													CoorFinaleLado_Pri0_Des180[NuPieza_B].LadoB.CoordenadaFinale_X := Supporto.XDim/2 + Supporto.OFSDE_X180;;
													CoorFinaleLado_Pri0_Des180[NuPieza_B].LadoB.CoordenadaFinale_Y := YEsternoLastra_A_B[NuPieza_B].Lado_B_180Grados + Supporto.OFSDE_Y0;
													CoorFinaleLado_Pri0_Des180[NuPieza_B].LadoB.CoordenadaFinale_Z := ZEsternoLastra_A_B[NuPieza_B].Lado_B_180Grados + Supporto.OFSDE_Z0;
													CoorFinaleLado_Pri0_Des180[NuPieza_B].LadoB.CoordenadaFinale_J := AlgoloAlfa_gradi + Supporto.OFSDE_J0 ;
											END_CASE
										4:	
											CASE LadoRegistarFor OF
												0: 
													CoorFinaleLado_Pri0_Des180[NuPieza_A].LadoA.CoordenadaFinale_X := Supporto.XDim/2 + Supporto.OFSDE_X0;;
													CoorFinaleLado_Pri0_Des180[NuPieza_A].LadoA.CoordenadaFinale_Y := YCoordinataAppoggioLastra_A_B[NuPieza_A].Lado_A_0Grados + Supporto.OFSDE_Y0;
													CoorFinaleLado_Pri0_Des180[NuPieza_A].LadoA.CoordenadaFinale_Z := ZCoordinataAppoggioLastra_A_B[NuPieza_A].Lado_A_0Grados + Supporto.OFSDE_Z0;
													CoorFinaleLado_Pri0_Des180[NuPieza_A].LadoA.CoordenadaFinale_J := AlgoloAlfa_gradi + Supporto.OFSDE_J0 ;
												180 :
													 
													CoorFinaleLado_Pri0_Des180[NuPieza_B].LadoB.CoordenadaFinale_X := Supporto.XDim/2 + Supporto.OFSDE_X180;;
													CoorFinaleLado_Pri0_Des180[NuPieza_B].LadoB.CoordenadaFinale_Y := YCoordinataAppoggioLastra_A_B[NuPieza_B].Lado_B_180Grados + Supporto.OFSDE_Y0;
													CoorFinaleLado_Pri0_Des180[NuPieza_B].LadoB.CoordenadaFinale_Z := ZCoordinataAppoggioLastra_A_B[NuPieza_B].Lado_B_180Grados + Supporto.OFSDE_Z0;
													CoorFinaleLado_Pri0_Des180[NuPieza_B].LadoB.CoordenadaFinale_J := AlgoloAlfa_gradi + Supporto.OFSDE_J0 ;
											END_CASE
																					
								END_CASE
										
						END_IF
					END_FOR
					
{endregion}

{Region "Ordinamento consecutivo prima un lato poi l'altro"}


		(* Ordinamento consecutivo prima un lato poi l'altro *)
		2:
			FOR Contador :=1 TO numeroLastre_int BY 1 DO
				Fun_PiezaLadoCaballete(Nu_PiezaGlobal:= Contador , Grados:= ADR(LadoRegistarFor)  ,
										 Nu_pieza_LadoA=>NuPieza_A , Nu_pieza_LadoB=> NuPieza_B  );
				IF NOT CalculoEstacionPickinPiezasDiferentes THEN 
					CASE TipoRisultato OF 
							1:	
								
								CoorFinaleLado_Pri0_Des180[Contador].LadoA.CoordenadaFinale_Y := YInternoLastra[Contador] + Supporto.OFSDE_Y0;
								CoorFinaleLado_Pri0_Des180[Contador].LadoA.CoordenadaFinale_Z := ZInternoLastra[Contador] + Supporto.OFSDE_Z0;
								
								CoorFinaleLado_Pri0_Des180[Contador].LadoB.CoordenadaFinale_Y := -YInternoLastra[Contador] + Supporto.OFSDE_Y180;
								CoorFinaleLado_Pri0_Des180[Contador].LadoB.CoordenadaFinale_Z := ZInternoLastra[Contador] + Supporto.OFSDE_Z180;
								
									
	
							2:
								CoorFinaleLado_Pri0_Des180[Contador].LadoA.CoordenadaFinale_Y := YCentroLastra[Contador] + Supporto.OFSDE_Y0;
								CoorFinaleLado_Pri0_Des180[Contador].LadoA.CoordenadaFinale_Z := ZCentroLastra[Contador] + Supporto.OFSDE_Z0;
								
								CoorFinaleLado_Pri0_Des180[Contador].LadoB.CoordenadaFinale_Y := -YCentroLastra[Contador] + Supporto.OFSDE_Y180;
								CoorFinaleLado_Pri0_Des180[Contador].LadoB.CoordenadaFinale_Z := ZCentroLastra[Contador] + Supporto.OFSDE_Z180;
							
							3:
								CoorFinaleLado_Pri0_Des180[Contador].LadoA.CoordenadaFinale_Y := YEsternoLastra[Contador] + Supporto.OFSDE_Y0;
								CoorFinaleLado_Pri0_Des180[Contador].LadoA.CoordenadaFinale_Z := ZEsternoLastra[Contador] + Supporto.OFSDE_Z0;
								
								CoorFinaleLado_Pri0_Des180[Contador].LadoB.CoordenadaFinale_Y := -YEsternoLastra[Contador] + Supporto.OFSDE_Y180;
								CoorFinaleLado_Pri0_Des180[Contador].LadoB.CoordenadaFinale_Z := ZEsternoLastra[Contador] + Supporto.OFSDE_Z180;
							
							4:
								CoorFinaleLado_Pri0_Des180[Contador].LadoA.CoordenadaFinale_Y := YCoordinataAppoggioLastra[Contador] + Supporto.OFSDE_Y0;
								CoorFinaleLado_Pri0_Des180[Contador].LadoA.CoordenadaFinale_Z := ZEsternoLastra[Contador] + Supporto.OFSDE_Z0;
								
								CoorFinaleLado_Pri0_Des180[Contador].LadoB.CoordenadaFinale_Y := -YCoordinataAppoggioLastra[Contador] + Supporto.OFSDE_Y180;
								CoorFinaleLado_Pri0_Des180[Contador].LadoB.CoordenadaFinale_Z := ZEsternoLastra[Contador] + Supporto.OFSDE_Z180;
	
					END_CASE
					CoorFinaleLado_Pri0_Des180[Contador].LadoA.CoordenadaFinale_X := Supporto.XDim/2 + Supporto.OFSDE_X180;
					CoorFinaleLado_Pri0_Des180[Contador].LadoA.CoordenadaFinale_J :=  AlgoloAlfa_gradi + Supporto.OFSDE_J0;
					CoorFinaleLado_Pri0_Des180[Contador].LadoB.CoordenadaFinale_J := 180 - AlgoloAlfa_gradi + Supporto.OFSDE_J180;
				ELSIF  CalculoEstacionPickinPiezasDiferentes AND Supporto.Tipologia = CAVALLETTO  THEN 	
					
					CASE TipoRisultato OF
						1:
							CASE LadoRegistarFor OF
								0:
									CoorFinaleLado_Pri0_Des180[NuPieza_A].LadoA.CoordenadaFinale_X := Supporto.XDim/2 + Supporto.OFSDE_X180;
									CoorFinaleLado_Pri0_Des180[NuPieza_A].LadoA.CoordenadaFinale_Y := YInternoLastra_A_B[NuPieza_A].Lado_A_0Grados + Supporto.OFSDE_Y0;
									CoorFinaleLado_Pri0_Des180[NuPieza_A].LadoA.CoordenadaFinale_Z := ZInternoLastra_A_B[NuPieza_A].Lado_A_0Grados + Supporto.OFSDE_Z0;
									CoorFinaleLado_Pri0_Des180[NuPieza_A].LadoA.CoordenadaFinale_J := AlgoloAlfa_gradi + Supporto.OFSDE_J0;
									
								180:
									CoorFinaleLado_Pri0_Des180[NuPieza_B].LadoA.CoordenadaFinale_X := Supporto.XDim/2 + Supporto.OFSDE_X180;
									CoorFinaleLado_Pri0_Des180[NuPieza_B].LadoB.CoordenadaFinale_Y := -YInternoLastra_A_B[NuPieza_B].Lado_B_180Grados + Supporto.OFSDE_Y180;
									CoorFinaleLado_Pri0_Des180[NuPieza_B].LadoB.CoordenadaFinale_Z := ZInternoLastra_A_B[NuPieza_B].Lado_B_180Grados + Supporto.OFSDE_Z180;
									CoorFinaleLado_Pri0_Des180[NuPieza_B].LadoB.CoordenadaFinale_J := 180 - AlgoloAlfa_gradi + Supporto.OFSDE_J180;
							END_CASE
						
						
						2:
							CASE LadoRegistarFor OF
								0:
									CoorFinaleLado_Pri0_Des180[NuPieza_A].LadoA.CoordenadaFinale_X := Supporto.XDim/2 + Supporto.OFSDE_X180;
									CoorFinaleLado_Pri0_Des180[NuPieza_A].LadoA.CoordenadaFinale_Y := YCentroLastra_A_B[NuPieza_A].Lado_A_0Grados + Supporto.OFSDE_Y0;
									CoorFinaleLado_Pri0_Des180[NuPieza_A].LadoA.CoordenadaFinale_Z := ZCentroLastra_A_B[NuPieza_A].Lado_A_0Grados + Supporto.OFSDE_Z0;
									CoorFinaleLado_Pri0_Des180[NuPieza_A].LadoA.CoordenadaFinale_J := AlgoloAlfa_gradi + Supporto.OFSDE_J0;
								180:
									CoorFinaleLado_Pri0_Des180[NuPieza_B].LadoA.CoordenadaFinale_X := Supporto.XDim/2 + Supporto.OFSDE_X180;
									CoorFinaleLado_Pri0_Des180[NuPieza_B].LadoB.CoordenadaFinale_Y := -YCentroLastra_A_B[NuPieza_B].Lado_B_180Grados + Supporto.OFSDE_Y180;
									CoorFinaleLado_Pri0_Des180[NuPieza_B].LadoB.CoordenadaFinale_Z := ZCentroLastra_A_B[NuPieza_B].Lado_B_180Grados + Supporto.OFSDE_Z180;
									CoorFinaleLado_Pri0_Des180[NuPieza_B].LadoB.CoordenadaFinale_J := 180 - AlgoloAlfa_gradi + Supporto.OFSDE_J180;
							END_CASE
						3:
							CASE LadoRegistarFor OF
								0:
									CoorFinaleLado_Pri0_Des180[NuPieza_A].LadoA.CoordenadaFinale_X := Supporto.XDim/2 + Supporto.OFSDE_X180;
									CoorFinaleLado_Pri0_Des180[NuPieza_A].LadoA.CoordenadaFinale_Y := YEsternoLastra_A_B[NuPieza_A].Lado_A_0Grados + Supporto.OFSDE_Y0;
									CoorFinaleLado_Pri0_Des180[NuPieza_A].LadoA.CoordenadaFinale_Z := ZEsternoLastra_A_B[NuPieza_A].Lado_A_0Grados + Supporto.OFSDE_Z0;
									CoorFinaleLado_Pri0_Des180[NuPieza_A].LadoA.CoordenadaFinale_J := AlgoloAlfa_gradi + Supporto.OFSDE_J0;
								180:
									CoorFinaleLado_Pri0_Des180[NuPieza_B].LadoA.CoordenadaFinale_X := Supporto.XDim/2 + Supporto.OFSDE_X180;
									CoorFinaleLado_Pri0_Des180[NuPieza_B].LadoB.CoordenadaFinale_Y := -YEsternoLastra_A_B[NuPieza_B].Lado_B_180Grados + Supporto.OFSDE_Y180;
									CoorFinaleLado_Pri0_Des180[NuPieza_B].LadoB.CoordenadaFinale_Z := ZEsternoLastra_A_B[NuPieza_B].Lado_B_180Grados + Supporto.OFSDE_Z180;
									CoorFinaleLado_Pri0_Des180[NuPieza_B].LadoB.CoordenadaFinale_J := 180 - AlgoloAlfa_gradi + Supporto.OFSDE_J180;
							END_CASE
						4:
							CASE LadoRegistarFor OF
								0:
									CoorFinaleLado_Pri0_Des180[NuPieza_A].LadoA.CoordenadaFinale_X := Supporto.XDim/2 + Supporto.OFSDE_X180;
									CoorFinaleLado_Pri0_Des180[NuPieza_A].LadoA.CoordenadaFinale_Y := YCoordinataAppoggioLastra_A_B[NuPieza_A].Lado_A_0Grados + Supporto.OFSDE_Y0;
									CoorFinaleLado_Pri0_Des180[NuPieza_A].LadoA.CoordenadaFinale_Z := ZEsternoLastra_A_B[NuPieza_A].Lado_A_0Grados + Supporto.OFSDE_Z0;
									CoorFinaleLado_Pri0_Des180[NuPieza_A].LadoA.CoordenadaFinale_J := AlgoloAlfa_gradi + Supporto.OFSDE_J0;
								180:
									CoorFinaleLado_Pri0_Des180[NuPieza_B].LadoA.CoordenadaFinale_X := Supporto.XDim/2 + Supporto.OFSDE_X180;
									CoorFinaleLado_Pri0_Des180[NuPieza_B].LadoB.CoordenadaFinale_Y := -YCoordinataAppoggioLastra_A_B[NuPieza_B].Lado_B_180Grados + Supporto.OFSDE_Y180;
									CoorFinaleLado_Pri0_Des180[NuPieza_B].LadoB.CoordenadaFinale_Z := ZEsternoLastra_A_B[NuPieza_B].Lado_B_180Grados + Supporto.OFSDE_Z180;
									CoorFinaleLado_Pri0_Des180[NuPieza_B].LadoB.CoordenadaFinale_J := 180 - AlgoloAlfa_gradi + Supporto.OFSDE_J180;
							END_CASE
						
						
						
						
						
					END_CASE
				
				END_IF
				END_FOR
		3:
			FOR Contador:=1 TO numeroLastre_int BY 1 DO
				XFinaleLado_0Grados[Contador] := Supporto.XDim/2 + Supporto.OFSDE_X0;
				CoorFinaleLado_Pri0_Des180[Contador].LadoA.CoordenadaFinale_X := XFinaleLado_0Grados[Contador];
					IF  NOT CalculoEstacionPickinPiezasDiferentes	THEN	
						CASE TipoRisultato OF
							1:	
								YFinaleLado_0Grados[Contador] := YInternoLastra[Contador] + Supporto.OFSDE_Y0;
								ZFinaleLado_0Grados[Contador] := ZInternoLastra[Contador] + Supporto.OFSDE_Z0;
								
							2:	
								YFinaleLado_0Grados[Contador] := YCentroLastra[Contador] + Supporto.OFSDE_Y0;
								ZFinaleLado_0Grados[Contador] := ZCentroLastra[Contador] + Supporto.OFSDE_Z0;
							3:	
								YFinaleLado_0Grados[Contador] := YEsternoLastra[Contador] + Supporto.OFSDE_Y0;
								ZFinaleLado_0Grados[Contador] := ZEsternoLastra[Contador] + Supporto.OFSDE_Z0;
							4:	
								YFinaleLado_0Grados[Contador] := YCoordinataAppoggioLastra[Contador] + Supporto.OFSDE_Y0;
								ZFinaleLado_0Grados[Contador] := ZEsternoLastra[Contador] + Supporto.OFSDE_Z0;
						END_CASE
					ELSIF CalculoEstacionPickinPiezasDiferentes	THEN
						CASE TipoRisultato OF
							1:	
								YFinaleLado_0Grados[Contador] := YInternoLastra_A_B[Contador].Lado_A_0Grados + Supporto.OFSDE_Y0;
								ZFinaleLado_0Grados[Contador] := ZInternoLastra_A_B[Contador].Lado_A_0Grados + Supporto.OFSDE_Z0;	
								
							2:	
								
								YFinaleLado_0Grados[Contador] := YCentroLastra_A_B[Contador].Lado_A_0Grados + Supporto.OFSDE_Y0;
								ZFinaleLado_0Grados[Contador] := ZCentroLastra_A_B[Contador].Lado_A_0Grados + Supporto.OFSDE_Z0;
							3:	
								YFinaleLado_0Grados[Contador] := YEsternoLastra_A_B[Contador].Lado_A_0Grados + Supporto.OFSDE_Y0;
								ZFinaleLado_0Grados[Contador] := ZEsternoLastra_A_B[Contador].Lado_A_0Grados + Supporto.OFSDE_Z0;
							4:	
								YFinaleLado_0Grados[Contador] := YCoordinataAppoggioLastra_A_B[Contador].Lado_A_0Grados + Supporto.OFSDE_Y0;
								ZFinaleLado_0Grados[Contador] := ZEsternoLastra_A_B[Contador].Lado_A_0Grados + Supporto.OFSDE_Z0;
						END_CASE
						CoorFinaleLado_Pri0_Des180[Contador].LadoA.CoordenadaFinale_Y := YFinaleLado_0Grados[Contador];	
						CoorFinaleLado_Pri0_Des180[Contador].LadoA.CoordenadaFinale_Z := ZFinaleLado_0Grados[Contador] ;
					END_IF
				
				JFinaleLado_0Grados[Contador] := AlgoloAlfa_gradi + Supporto.OFSDE_J0;
				CoorFinaleLado_Pri0_Des180[Contador].LadoA.CoordenadaFinale_J := JFinaleLado_0Grados[Contador] ;
			END_FOR	
		IF  CalculoEstacionPickinPiezasDiferentes OR NOT  HabiCalTodasCordenadas  THEN
				XFinale := 	XFinaleLado_0Grados ;	
				YFinale := 	YFinaleLado_0Grados ;
				ZFinale := 	ZFinaleLado_0Grados ;
				JFinale := 	JFinaleLado_0Grados ;	
		END_IF		
				
	4:
		FOR Contador:=1 TO numeroLastre_int BY 1 DO
						
			XFinaleLado_180Grados[Contador] := Supporto.XDim/2 + Supporto.OFSDE_X180;
			
				IF  NOT CalculoEstacionPickinPiezasDiferentes	THEN	
					CASE TipoRisultato OF
						1:	
							YFinaleLado_180Grados[Contador] := -YInternoLastra[Contador] + Supporto.OFSDE_Y180;
							ZFinaleLado_180Grados[Contador] := ZInternoLastra[Contador] + Supporto.OFSDE_Z180;
							
						2:	
							YFinaleLado_180Grados[Contador] := -YCentroLastra[Contador] + Supporto.OFSDE_Y180;
							ZFinaleLado_180Grados[Contador] := ZCentroLastra[Contador] + Supporto.OFSDE_Z180;
						3:	
							YFinaleLado_180Grados[Contador] := -YEsternoLastra[Contador] + Supporto.OFSDE_Y180;
							ZFinaleLado_180Grados[Contador] := ZEsternoLastra[Contador] + Supporto.OFSDE_Z180;
						4:	
							YFinaleLado_180Grados[Contador] := -YCoordinataAppoggioLastra[Contador] + Supporto.OFSDE_Y180;
							ZFinaleLado_180Grados[Contador] := ZEsternoLastra[Contador] + Supporto.OFSDE_Z180;
					END_CASE
				ELSIF CalculoEstacionPickinPiezasDiferentes	THEN
					CASE TipoRisultato OF
						1:	
							YFinaleLado_180Grados[Contador] := -YInternoLastra_A_B[Contador].Lado_B_180Grados + Supporto.OFSDE_Y180;
							ZFinaleLado_180Grados[Contador] := ZInternoLastra_A_B[Contador].Lado_B_180Grados + Supporto.OFSDE_Z180;	
							
						2:	
							
							YFinaleLado_180Grados[Contador] := -YCentroLastra_A_B[Contador].Lado_B_180Grados + Supporto.OFSDE_Y180;
							ZFinaleLado_180Grados[Contador] := ZCentroLastra_A_B[Contador].Lado_B_180Grados + Supporto.OFSDE_Z180;
						3:	
							YFinaleLado_180Grados[Contador] := -YEsternoLastra_A_B[Contador].Lado_B_180Grados + Supporto.OFSDE_Y180;
							ZFinaleLado_180Grados[Contador] := ZEsternoLastra_A_B[Contador].Lado_B_180Grados + Supporto.OFSDE_Z180;
						4:	
							YFinaleLado_180Grados[Contador] := -YCoordinataAppoggioLastra_A_B[Contador].Lado_B_180Grados + Supporto.OFSDE_Y180;
							ZFinaleLado_180Grados[Contador] := ZEsternoLastra_A_B[Contador].Lado_B_180Grados + Supporto.OFSDE_Z180;
							
					END_CASE
					CoorFinaleLado_Pri0_Des180[Contador].LadoB.CoordenadaFinale_Y := YFinaleLado_180Grados[Contador] ;
					CoorFinaleLado_Pri0_Des180[Contador].LadoB.CoordenadaFinale_Z := ZFinaleLado_180Grados[Contador] ;
				END_IF
			
			JFinaleLado_180Grados[Contador] := 180 - AlgoloAlfa_gradi + Supporto.OFSDE_J180; 
			CoorFinaleLado_Pri0_Des180[Contador].LadoB.CoordenadaFinale_J := JFinaleLado_180Grados[Contador] ;
		END_FOR		
	
		IF  CalculoEstacionPickinPiezasDiferentes OR NOT  HabiCalTodasCordenadas  THEN
				XFinale := 	XFinaleLado_180Grados ;	
				YFinale := 	YFinaleLado_180Grados ;
				ZFinale := 	ZFinaleLado_180Grados ;
				JFinale := 	JFinaleLado_180Grados ;	
		END_IF	
END_CASE
				
END_FOR
		













{endregion}
	
		
		
		
			(* Calcolo delle coordinate X,Y,Z,J del punto finale sulla base del TipoRisultato *)
		(*	Fb_CalculoFormaciones(
				TipoCalForCavallete:= CalForCavallete , 
				numeroLastre_int:= numeroLastre_int , 
				TipoRisultato:=TipoRisultato  , 
				AlgoloAlfa_gradi:= AlgoloAlfa_gradi , 
				CalculoEstacionPickinPiezasDiferentes:= CalculoEstacionPickinPiezasDiferentes , 
				Supporto:= ADR(Supporto), 
				XFinale:=  ADR(XFinale) , 
				CoorFinaleLado_Pri0_Des180:=  ADR(CoorFinaleLado_Pri0_Des180) , 
				YFinale:=  ADR(YFinale) , 
				YInternoLastra:=  ADR(YInternoLastra) , 
				YCentroLastra:=  ADR(YCentroLastra) , 
				YEsternoLastra:=  ADR(YEsternoLastra), 
				YCoordinataAppoggioLastra:=  ADR(YCoordinataAppoggioLastra), 
				ZFinale:= ADR(ZFinale) , 
				ZInternoLastra:=  ADR(ZInternoLastra) , 
				ZCentroLastra:=  ADR(ZCentroLastra) , 
				ZEsternoLastra:= ADR(ZEsternoLastra) , 
				JFinale:=  ADR(JFinale) , 
				XInternoLastra_A_B:=  ADR(XInternoLastra_A_B) , 
				YInternoLastra_A_B:=  ADR(YInternoLastra_A_B) , 
				ZInternoLastra_A_B:=  ADR(ZInternoLastra_A_B) , 
				XCentroLastra_A_B:=  ADR(XCentroLastra_A_B) , 
				YCentroLastra_A_B:=  ADR(YCentroLastra_A_B) , 
				ZCentroLastra_A_B:=  ADR(ZCentroLastra_A_B) , 
				XEsternoLastra_A_B:=  ADR(XEsternoLastra_A_B) , 
				YEsternoLastra_A_B:=  ADR(YEsternoLastra_A_B) , 
				ZEsternoLastra_A_B:=  ADR(ZEsternoLastra_A_B) , 
				YCoordinataAppoggioLastra_A_B:=  ADR(YCoordinataAppoggioLastra_A_B) , 
				ZCoordinataAppoggioLastra_A_B:=  ADR(ZCoordinataAppoggioLastra_A_B) );
		*)
	(*
		Fb_CalculoFormacionesTodo0_grados(
			CalculoEstacionPickinPiezasDiferentes:= CalculoEstacionPickinPiezasDiferentes , 
			numeroLastre_int:= numeroLastre_int , 
			TipoCalForCavallete:= CalForCavallete , 
			TipoRisultato:=TipoRisultato , 
			AlgoloAlfa_gradi:= AlgoloAlfa_gradi, 
			Supporto:= ADR(Supporto) , 
			YCoordinataAppoggioLastra:= ADR(YCoordinataAppoggioLastra) , 
			ZCoordinataAppoggioLastra:= ADR(ZCoordinataAppoggioLastra), 
			YCoordinataAppoggioLastra_A_B:=ADR(YCoordinataAppoggioLastra_A_B) , 
			ZCoordinataAppoggioLastra_A_B:=ADR(ZCoordinataAppoggioLastra_A_B) , 
			XFinaleLado_0Grados:= ADR(XFinaleLado_0Grados) , 
			YFinaleLado_0Grados:= ADR(YFinaleLado_0Grados), 
			ZFinaleLado_0Grados:=ADR(ZFinaleLado_0Grados) , 
			JFinaleLado_0Grados:= ADR(JFinaleLado_0Grados) , 
			XInternoLastra:=ADR(XInternoLastra) , 
			YInternoLastra:=ADR(YInternoLastra) , 
			ZInternoLastra:=ADR(ZInternoLastra) , 
			XCentroLastra:=ADR(XCentroLastra) , 
			YCentroLastra:= ADR(YCentroLastra), 
			ZCentroLastra:= ADR(ZCentroLastra), 
			XEsternoLastra:=ADR(XEsternoLastra) , 
			YEsternoLastra:= ADR(YEsternoLastra), 
			ZEsternoLastra:= ADR(ZEsternoLastra) , 
			XInternoLastra_A_B:= ADR(XInternoLastra_A_B), 
			YInternoLastra_A_B:= ADR(YInternoLastra_A_B) , 
			ZInternoLastra_A_B:= ADR(ZInternoLastra_A_B) , 
			XCentroLastra_A_B:= ADR(XCentroLastra_A_B) , 
			YCentroLastra_A_B:= ADR(YCentroLastra_A_B) , 
			ZCentroLastra_A_B:= ADR(ZCentroLastra_A_B) , 
			XEsternoLastra_A_B:= ADR(XEsternoLastra_A_B) , 
			YEsternoLastra_A_B:= ADR(YEsternoLastra_A_B) , 
			ZEsternoLastra_A_B:= ADR(YEsternoLastra_A_B) );	
			
		*)
		(*
		Fb_CalculoFormacionesTodo180_grados(
			CalculoEstacionPickinPiezasDiferentes:= CalculoEstacionPickinPiezasDiferentes , 
			numeroLastre_int:= numeroLastre_int , 
			TipoCalForCavallete:= CalForCavallete , 
			TipoRisultato:= TipoRisultato , 
			AlgoloAlfa_gradi:= AlgoloAlfa_gradi , 
			Supporto:= ADR(Supporto), 
			YCoordinataAppoggioLastra:= ADR(YCoordinataAppoggioLastra) , 
			ZCoordinataAppoggioLastra:=ADR(ZCoordinataAppoggioLastra) , 
			YCoordinataAppoggioLastra_A_B:= ADR(YCoordinataAppoggioLastra_A_B) , 
			ZCoordinataAppoggioLastra_A_B:= ADR(ZCoordinataAppoggioLastra_A_B) , 
			XFinaleLado_180Grados:= ADR(XFinaleLado_180Grados) , 
			YFinaleLado_180Grados:= ADR(YFinaleLado_180Grados) , 
			ZFinaleLado_180Grados:= ADR(ZFinaleLado_180Grados) , 
			JFinaleLado_180Grados:= ADR(JFinaleLado_180Grados) , 
			XInternoLastra:= ADR(XInternoLastra) , 
			YInternoLastra:= ADR(YInternoLastra) , 
			ZInternoLastra:=ADR(ZInternoLastra) , 
			XCentroLastra:= ADR(XCentroLastra) , 
			YCentroLastra:= ADR(YCentroLastra), 
			ZCentroLastra:= ADR(ZCentroLastra) , 
			XEsternoLastra:= ADR(XEsternoLastra) , 
			YEsternoLastra:= ADR(YEsternoLastra) , 
			ZEsternoLastra:= ADR(ZEsternoLastra) , 
			XInternoLastra_A_B:= ADR(XInternoLastra_A_B) , 
			YInternoLastra_A_B:= ADR(YInternoLastra_A_B) , 
			ZInternoLastra_A_B:= ADR(ZInternoLastra_A_B) , 
			XCentroLastra_A_B:= ADR(XCentroLastra_A_B) , 
			YCentroLastra_A_B:= ADR(YCentroLastra_A_B) , 
			ZCentroLastra_A_B:= ADR(ZCentroLastra_A_B) , 
			XEsternoLastra_A_B:= ADR(XEsternoLastra_A_B), 
			YEsternoLastra_A_B:=ADR(YEsternoLastra_A_B) , 
			ZEsternoLastra_A_B:=ADR(ZEsternoLastra_A_B) );		
			*)	
								



			
			// Alimentazione della struttura FormingSlab
			FOR counter1:=1 TO MAXFORMINGSLAB DO// numeroLastre_int*2 BY 1 DO
				IF counter1 <= numeroLastre_int THEN
					FormingSlab.Enable := 1;										// Abilitato
					//FormingSlab.Code[1] := 1;
					FormingSlab.PElement[counter1].Typology 			:= OrdineDepositoSxDx[counter1];
					FormingSlab.PElement[counter1].X 					:= XFinale[counter1];
					FormingSlab.PElement[counter1].XDim 				:= Materiale[OrdineDepositoSxDx[counter1]].XDim;		// Dimensione X Lastra
					FormingSlab.PElement[counter1].Y 					:= YFinale[counter1];
					FormingSlab.PElement[counter1].YDim 				:= Materiale[OrdineDepositoSxDx[counter1]].YDim;		// Dimensione Y Lastra
					FormingSlab.PElement[counter1].Z 					:= ZFinale[counter1];
					FormingSlab.PElement[counter1].ZDim 				:= Materiale[OrdineDepositoSxDx[counter1]].ZDim;		// Dimensione Z Lastra
					FormingSlab.PElement[counter1].J 					:= JFinale[counter1];
					
					FormingSlab.PElement[counter1].CooCavallete 		:= CoorFinaleLado_Pri0_Des180[counter1] ;
				ELSE
					FormingSlab.PElement[counter1].Typology := OrdineDepositoSxDx[counter1];
					FormingSlab.PElement[counter1].X 		:= -1;
					FormingSlab.PElement[counter1].XDim 	:= -1;	
					FormingSlab.PElement[counter1].Y 		:= -1;
					FormingSlab.PElement[counter1].YDim 	:= -1;		
					FormingSlab.PElement[counter1].Z 		:= -1;
					FormingSlab.PElement[counter1].ZDim 	:= -1;	
					FormingSlab.PElement[counter1].J 		:= -1;
				END_IF
			END_FOR		
		

		INCLINATO_LATOSINGOLO:		// Tipo deposito inclinato singolo lato (Bundle)
			numeroLastre_int := 0;
			FOR counter1:=1 TO MAXFORMINGSLAB/2 BY 1 DO
				IF (TipoElementoDep[counter1] > 0) THEN
				numeroLastre_int := numeroLastre_int+1;
				END_IF;
			END_FOR
	
			(* Controlli dati coerenti --- DA FARE --- *)
						
			(* calcolo angolo alfa dell'inclinazione appoggio della lastra *)
			AngoloAlfa_rad := deg_to_rad(Supporto.AngoloAlfaBundle); // Angolo superiore appoggio cavallina (in radianti)
			AlgoloAlfa_gradi := Supporto.AngoloAlfaBundle; 
			
			
			(* Calcolo angolo beta dell'eventuale piano di appoggio inclinato della cavallina*)
			AngoloBeta_rad := AngoloAlfa_rad; 	// Angolo del piano di appoggio inclinato della cavallina (in radianti)
			AngoloBeta_gradi := AlgoloAlfa_gradi;					// Angolo del piano di appoggio inclinato della cavallina (in gradi)
	
			
			// Calcolo lo spessore di ogni singola lastra/falda depositata sul lato della cavallina
			Spessore_Lastra_Inclinata[1] := 0;
			FOR counter2:=2 TO MAXFORMINGSLAB/2 BY 1 DO
				Spessore_Lastra_Inclinata[counter2] := Materiale[TipoElementoDep[counter2-1]].ZDim / COS(AngoloAlfa_rad);
			END_FOR;
			
			// Calcola lo spessore complessivo fino al passo n delle lastre/falde depositate sul singolo lato della cavallina 
			//memset(ADR(Spessore_Lastra_Inclinata_Cumulato), 0 , SIZEOF(Spessore_Lastra_Inclinata_Cumulato));
			
			IF (Spessore_Lastra_Inclinata_Cumulato[2] = 0) THEN
				FOR counter2:=1 TO MAXFORMINGSLAB/2 BY 1 DO
					FOR counter1 := 1 TO counter2 BY 1 DO
						Spessore_Lastra_Inclinata_Cumulato[counter2] := Spessore_Lastra_Inclinata_Cumulato[counter2]+Spessore_Lastra_Inclinata[counter1];
					END_FOR
				END_FOR
			END_IF
			
			// Numero di possibili lastre sul singolo lato
			FOR counter1:=1 TO MAXFORMINGSLAB/2 BY 1 DO
				IF (TipoElementoDep[counter1] > 0) AND ((Spessore_Lastra_Inclinata_Cumulato[counter1] >0) AND (Spessore_Lastra_Inclinata_Cumulato[counter1] < Supporto.DimBaseUtile)) THEN
					numeroLastre_int := counter1;
				END_IF
				IF (Spessore_Lastra_Inclinata_Cumulato[counter1] >= Supporto.DimBaseUtile) THEN
					Errore := ErrNumeroPezzi;	// il supervisore mi ha passato troppe lastre rispetto allo spazio utile
				END_IF
			END_FOR
			
			// Calcolo lo spostamento del punto centrale e del punto esterno della singola lastra/falda rispetto al punto interno(iniziale) della medesima lastra/falda
			FOR counter2:=1 TO numeroLastre_int BY 1 DO
				Yd1[counter2] := Materiale[TipoElementoDep[counter2]].ZDim / 2 * COS (AngoloAlfa_rad);		// Spostamento Centro lastra da interno lastra in Y
				Zd1[counter2] := Materiale[TipoElementoDep[counter2]].ZDim / 2 * SIN (AngoloAlfa_rad);		// Spostamento Centro lastra da interno lastra in Z
				Yd2[counter2] := Materiale[TipoElementoDep[counter2]].ZDim  * COS (AngoloAlfa_rad);			// Spostamento esterno lastra da interno lastra in Y
				Zd2[counter2] := Materiale[TipoElementoDep[counter2]].ZDim  * SIN (AngoloAlfa_rad);			// Spostamento esterno lastra da interno lastra in Z
			END_FOR
			
			// Calcolo la proiezione mancante di ogni singola lastra/falda; Tramite CI posso calcolare lo spostamento Yd3,Zd3 dovuto al piano inclinato
			// dovuto all'angolo beta. Utilizzo il teorema dei seni per calcolare ogni CI da SLIC
			FOR counter1:=1 TO numeroLastre_int BY 1 DO
				CI[counter1] := (Spessore_Lastra_Inclinata_Cumulato[counter1] * SIN (AngoloBeta_rad));
				Yd3[counter1] := -CI[counter1] * SIN(AngoloAlfa_rad);
				Zd3[counter1] := CI[counter1] * COS(AngoloAlfa_rad);
			END_FOR;
			
			// Quota Y e Z del punto di appoggio di ogni lastra sulla cavallina
			// Quota Y e Z del punto interno centrale di ogni lastra; corrisponde a YInternoLastra e ZInternoLastra
			FOR counter2:=1 TO numeroLastre_int BY 1 DO
				XInternoLastra[counter2] := Supporto.XDim/2;
				YCoordinataAppoggioLastra[counter2] := Spessore_Lastra_Inclinata_Cumulato[counter2] + Yd3[counter2];
				YInternoLastra[counter2] := YCoordinataAppoggioLastra[counter2] - (Materiale[TipoElementoDep[counter2]].YDim / 2) * SIN (AngoloAlfa_rad);
				ZCoordinataAppoggioLastra[counter2] := Supporto.ZDim + Zd3[counter2];
				ZInternoLastra[counter2] := ZCoordinataAppoggioLastra[counter2] + (Materiale[TipoElementoDep[counter2]].YDim / 2) * COS (AngoloAlfa_rad); 
			END_FOR
	
			(* Calcolo delle coordinate X,Y,Z di ogni singola lastra/falda, centrale o esterno *)
			FOR counter2:=1 TO numeroLastre_int BY 1 DO
				XCentroLastra[counter2] := Supporto.XDim/2;
				YCentroLastra[counter2] := YInternoLastra[counter2] + Yd1[counter2];
				ZCentroLastra[counter2] := ZInternoLastra[counter2] + Zd1[counter2];
				
				XEsternoLastra[counter2] := Supporto.XDim/2;
				YEsternoLastra[counter2] := YInternoLastra[counter2] + Yd2[counter2];	
				ZEsternoLastra[counter2] := ZInternoLastra[counter2] + Zd2[counter2];
			END_FOR;
			
			(* Pulisco le uscite e setto a TERMINATORE tutti gli elementi di FormingSlab*)
			//memset(ADR(XFinale),0,SIZEOF(XFinale));memset(ADR(YFinale),0,SIZEOF(XFinale));memset(ADR(ZFinale),0,SIZEOF(XFinale));memset(ADR(JFinale),0,SIZEOF(XFinale));
			//memset(ADR(FormingSlab),0,SIZEOF(FormingSlab));
			FOR counter1 := 1 TO MAXFORMINGSLAB DO
				FormingSlab.PElement[counter1].Typology := TERMINATORE;
			END_FOR
			
			(* Calcolo delle coordinate X,Y,Z,J del punto finale sulla base del TipoRisultato *)
			FOR counter2:=1 TO numeroLastre_int BY 1 DO
				CASE supporto.LatoDeposito OF
					180:		// Lato DX della cavallina
						XFinale[counter2] := Supporto.XDim/2 + Supporto.OFSDE_X180;
						CASE TipoRisultato OF
							1:	
								YFinale[counter2] := -YInternoLastra[counter2] + Supporto.OFSDE_Y180;
								ZFinale[counter2] := ZInternoLastra[counter2] + Supporto.OFSDE_Z180;
							2:	
								YFinale[counter2] := -YCentroLastra[counter2] + Supporto.OFSDE_Y180;
								ZFinale[counter2] := ZCentroLastra[counter2] + Supporto.OFSDE_Z180;
							3:	
								YFinale[counter2] := -YEsternoLastra[counter2] + Supporto.OFSDE_Y180;
								ZFinale[counter2] := ZEsternoLastra[counter2] + Supporto.OFSDE_Z180;
						END_CASE
						JFinale[counter2] := 180 - AlgoloAlfa_gradi + Supporto.OFSDE_J180; 
					0:	// Lato SX della cavallina
						XFinale[counter2] := Supporto.XDim/2 + Supporto.OFSDE_X0;
						CASE TipoRisultato OF
							1:	
								YFinale[counter2] := YInternoLastra[counter2] + Supporto.OFSDE_Y0;
								ZFinale[counter2] := ZInternoLastra[counter2] + Supporto.OFSDE_Z0;
							2:	
								YFinale[counter2] := YCentroLastra[counter2] + Supporto.OFSDE_Y0;
								ZFinale[counter2] := ZCentroLastra[counter2] + Supporto.OFSDE_Z0;
							3:	
								YFinale[counter2] := YEsternoLastra[counter2] + Supporto.OFSDE_Y0;
								ZFinale[counter2] := ZEsternoLastra[counter2] + Supporto.OFSDE_Z0;
						END_CASE
						JFinale[counter2] := AlgoloAlfa_gradi + Supporto.OFSDE_J0;
				END_CASE

				
				// Alimentazione della struttura FormingSlab
				FOR counter1:=1 TO numeroLastre_int BY 1 DO
					FormingSlab.Enable := 1;										// Abilitato
					FormingSlab.Code[1] := 1;
					FormingSlab.PElement[counter1].Typology := Materiale[OrdineDepositoSxDx[counter1]].Typology;
					FormingSlab.PElement[counter1].X := XFinale[counter1];
					FormingSlab.PElement[counter1].XDim := Materiale[OrdineDepositoSxDx[counter1]].XDim;		// Dimensione X Lastra
					FormingSlab.PElement[counter1].Y := YFinale[counter1];
					FormingSlab.PElement[counter1].YDim := Materiale[OrdineDepositoSxDx[counter1]].YDim;		// Dimensione Y Lastra
					FormingSlab.PElement[counter1].Z := ZFinale[counter1];
					FormingSlab.PElement[counter1].ZDim := Materiale[OrdineDepositoSxDx[counter1]].ZDim;		// Dimensione Z Lastra
					FormingSlab.PElement[counter1].J := JFinale[counter1];
				END_FOR		
			END_FOR;	
	END_CASE


	// Salvataggio su file della Formatura 
	{region "Salvataggio File Formatura"}
	P_TextModeWrite.database[0,0] := 'X Finale';
	P_TextModeWrite.database[0,1] := 'Y Finale';
	P_TextModeWrite.database[0,2] := 'Z Finale';
	P_TextModeWrite.database[0,3] := 'J Finale';
	CASE TipoDeposito OF
		ORIZZONTALE :	
			P_TextModeWrite.database[0,4] := 'ORIZZONTALE';
			P_TextModeWrite.database[0,5] := UINT_TO_STRING(numeroLastre_int);
		INCLINATO : 
			P_TextModeWrite.database[0,4] := 'INCLINATO';
			P_TextModeWrite.database[0,5] := UINT_TO_STRING(numeroLastre_int*2);
		INCLINATO_LATOSINGOLO :
			P_TextModeWrite.database[0,4] := 'INCLINATO_LATOSINGOLO';
			P_TextModeWrite.database[0,5] := UINT_TO_STRING(numeroLastre_int);	  
	END_CASE
	CASE TipoRisultato OF
		1:	P_TextModeWrite.database[0,6] := 'PUNTO INTERNO';
		2:	P_TextModeWrite.database[0,6] := 'PUNTO CENTRALE';
		3:	P_TextModeWrite.database[0,6] := 'PUNTO ESTERNO';
	END_CASE
	
	FOR counter1 :=1 TO MAXFORMINGSLAB DO
		P_TextModeWrite.database[counter1,0] := LREAL_TO_STRING(XFinale[counter1]);
		P_TextModeWrite.database[counter1,1] := LREAL_TO_STRING(YFinale[counter1]);
		P_TextModeWrite.database[counter1,2] := LREAL_TO_STRING(ZFinale[counter1]);
		P_TextModeWrite.database[counter1,3] := LREAL_TO_STRING(JFinale[counter1]);
	END_FOR
	
	CASE TipoDeposito OF	// Numero di righe da scrivere sul file a seconda che sia CASSA o CAVALLINA
		ORIZZONTALE :	
			P_TextModeWrite.num_Row := numeroLastre_int;
		INCLINATO : 
			P_TextModeWrite.num_Row := numeroLastre_int * 2;
		INCLINATO_LATOSINGOLO : 
			P_TextModeWrite.num_Row := numeroLastre_int;
	END_CASE
	
	{endregion}
	CalcolaFormaturaDone := TRUE;	
	P_TextModeWrite.bWrite := TRUE; //Scrivo log per calcoli
ELSIF NOT CalcolaFormatura AND CalcolaFormaturaDone THEN
	CalcolaFormaturaDone := FALSE;
END_IF

//chiamata fb per log calcoli	
//___________P_TextModeWrite();
IF P_TextModeWrite.bWriteDone AND P_TextModeWrite.bWrite THEN
	P_TextModeWrite.bWrite := FALSE; 
END_IF

END_FUNCTION_BLOCK

// ---- POUs/TFPalletizerData_Lastre/Formatura/Utility/CSV read_write in text mode/P_TextModeWrite.TcPOU
(* Writing of CSV file in text mode. None of the field value is containing any non-printing control characters like line feed, carriage return, quotation marks, semicolon... *)
FUNCTION_BLOCK P_TextModeWrite
VAR_INPUT
	bWrite			: BOOL;(* Rising edge starts program execution *)
	database		: ARRAY[0..MAX_CSV_ROWS, 0..MAX_CSV_COLUMNS ] OF STRING(MAX_CSV_FIELD_LENGTH); (* Source PLC database *)
	num_Row 		: UINT;	// Numero di righe da scrivere sul file
END_VAR

VAR_OUTPUT
	bWriteDone 		: BOOL := FALSE;	// External output to know when the FB is executed
END_VAR

VAR	
	sNetId			: T_AmsNetId := '';	(* TwinCAT system network address *)
	sFileName		: T_MaxString := 'C:\CSVData\TextModeGen.csv';(* CSV destination file path and name *)
	sCSVLine		: T_MaxString := '';(* Single CSV text line (row, record), we are using string as record buffer (your are able to see created fields) *)
	sCSVField		: T_MaxString := '';(* Single CSV field value (column, record field) *)
	bBusy			: BOOL;
	bError			: BOOL;
	nErrId			: UDINT;
	nRow	 		: UDINT 	:= 0;(* Row number (record) *)
	nColumn			: UDINT 	:= 0;(* Column number (record field) *)
	hFile			: UINT		:= 0;(* File handle of the source file *)
	step			: DWORD 	:= 0;
	fbFileOpen		: FB_FileOpen;(* Opens file *)
	fbFileClose		: FB_FileClose;(* Closes file *)
	fbFilePuts		: FB_FilePuts;(* Writes one record (line) *)
	fbWriter		: FB_CSVMemBufferWriter;(* Helper function block used to create CSV data bytes (single record line) *)
END_VAR
VAR CONSTANT
	MAX_CSV_ROWS 			: UDINT := 200;		// Numero massimo righe per file csv della formatura
	MAX_CSV_COLUMNS 		: UDINT := 10;		// Numero massimo colonne per file csv della formatura
	MAX_CSV_FIELD_LENGTH	: UDINT := 100;		// Dimensione massima campo CSV del file formatura
END_VAR

IF bWrite = TRUE THEN
	bWriteDone := FALSE;		// Inizio un nuovo ciclo di scrittura
END_IF


CASE step OF
	0:	(* Wait for rising edge at bWrite variable *)
		IF bWrite THEN
			bWrite 	:= FALSE;
			bBusy 	:= TRUE;
			bError	:= FALSE;
			nErrId	:= 0;
			hFile	:= 0;
			nRow	:= 0;
			nColumn	:= 0;
			step 	:= 1;
		END_IF

	1:	(* Open source file *)
		fbFileOpen(  bExecute := FALSE  );
		fbFileOpen( sNetId := sNetId, sPathName := sFileName, nMode := FOPEN_MODEWRITE OR FOPEN_MODETEXT,(* Open file in TEXT mode! *)
					ePath := PATH_GENERIC, bExecute := TRUE );
		step := 2;

	2:(* Wait until open not busy *)
		fbFileOpen( bExecute := FALSE, bError => bError, nErrID => nErrID, hFile => hFile );
		IF NOT fbFileOpen.bBusy THEN
			IF NOT fbFileOpen.bError THEN
				step := 3;
			ELSE(* Error: file not found? *)
				step := 100;
			END_IF
		END_IF

	3:(* Convert one PLC record to CSV format *)
		sCSVLine := '';
		fbWriter.eCmd := eEnumCmd_First;(* Write first field value *)
		IF nRow <= num_Row THEN

			FOR nColumn := 0 TO MAX_CSV_COLUMNS BY 1 DO

				sCSVField := STRING_TO_CSVFIELD( database[ nRow, nColumn ], FALSE );(* TODO: Get field value from your application *)

				(* Add new field to the record buffer *)
				fbWriter( 	pBuffer := ADR( sCSVLine ), cbBuffer := SIZEOF( sCSVLine ) - 1, putValue := sCSVField, pValue := 0, cbValue := 0,
							bCRLF := ( nColumn = MAX_CSV_COLUMNS ) );(* bCRLF == TRUE => Write CRLF after the last field value *)
				IF fbWriter.bOk THEN
					fbWriter.eCmd := eEnumCmd_Next;(* Write next field value *)
				ELSE(* Error *)
					step := 100;
					RETURN;
				END_IF

			END_FOR(* FOR nColumn := 0... *)

			(* FB_FilePuts adds allready CR (carriage return) to the written line.
			We have to replace the $R$L characters with $L character to avoid double CR. *)
			IF RIGHT( sCSVLine, 2 ) = '$R$L' THEN
				sCSVLine := REPLACE( sCSVLine, '$L', 2, LEN( sCSVLine ) - 1 );
			END_IF

			nRow := nRow + 1;(* Increment number of created records (rows) *)
			step := 4;(* Write record to the file *)

		ELSE(* All rows written => Close file *)
			step := 10;
		END_IF

	4:	(* Write single text line *)
		fbFilePuts( bExecute := FALSE );
		fbFilePuts( sNetId := sNetId, hFile := hFile, sLine := sCSVLine, bExecute := TRUE );
		step := 5;

	5:(* Wait until write not busy *)
		fbFilePuts( bExecute := FALSE, bError => bError, nErrID => nErrID );
		IF NOT fbFilePuts.bBusy THEN
			IF NOT fbFilePuts.bError THEN
				step := 3;(* Write next record *)
			ELSE(* Error *)
				step := 100;
			END_IF
		END_IF

	10:	(* Close source file *)
		fbFileClose( bExecute := FALSE );
		fbFileClose( sNetId := sNetId, hFile := hFile, bExecute := TRUE );
		step := 11;
		//step := 0;
		RETURN;

	11:(* Wait until close not busy *)
		fbFileClose( bExecute := FALSE, bError => bError, nErrID => nErrID );
		IF ( NOT fbFileClose.bBusy ) THEN
			hFile := 0;
			step := 100;
		END_IF

	100: (* Error or ready step => cleanup *)
		IF ( hFile <> 0 ) THEN
			step := 10; (* Close the source file *)
		ELSE
			bBusy := FALSE;
			bWriteDone := TRUE;
			step := 0;	(* Ready *)
		END_IF

END_CASE

END_FUNCTION_BLOCK

// ---- Data types/AlbertoPruevas/BloqueFunciones/CalculoFormaciones/Fb_CalculoCoordenadasFinalesFormacion.TcPOU
FUNCTION_BLOCK Fb_CalculoCoordenadasFinalesFormacion
VAR_INPUT
	TipoCalForCavallete 					: UINT ;
	numeroLastre_int 						: UINT ;
	TipoRisultato							: UINT ;
	AlgoloAlfa_gradi						: LREAL ;
	CalculoEstacionPickinPiezasDiferentes 	: BOOL ;
	Supporto 								: POINTER TO TFMachinePalletizer_Pallet;
	XFinale 								: POINTER TO  ARRAY [1..MAXFORMINGSLAB] OF LREAL;
	
	CoorFinaleLado_Pri0_Des180 : POINTER TO ARRAY [1..MAXFORMINGSLAB] OF Es_CoordenadasCaballeteLadoA_ladoB ;
	
	YFinale 					: POINTER TO  ARRAY [1..MAXFORMINGSLAB] OF LREAL;
	YInternoLastra 				: POINTER TO  ARRAY [1..MAXFORMINGSLAB] OF LREAL;
	YCentroLastra				: POINTER TO  ARRAY [1..MAXFORMINGSLAB] OF LREAL;
	YEsternoLastra				: POINTER TO  ARRAY [1..MAXFORMINGSLAB] OF LREAL;
	YCoordinataAppoggioLastra 	: POINTER TO  ARRAY [1..MAXFORMINGSLAB] OF LREAL;
	
	ZFinale 					: POINTER TO  ARRAY [1..MAXFORMINGSLAB] OF LREAL;
	ZInternoLastra				: POINTER TO  ARRAY [1..MAXFORMINGSLAB] OF LREAL;
	ZCentroLastra      			: POINTER TO  ARRAY [1..MAXFORMINGSLAB] OF LREAL;
	ZEsternoLastra				: POINTER TO  ARRAY [1..MAXFORMINGSLAB] OF LREAL;
	
	JFinale 					: POINTER TO  ARRAY [1..MAXFORMINGSLAB] OF LREAL;
	
	XInternoLastra_A_B : POINTER TO ARRAY [1..MAXFORMINGSLAB] OF ES_SpesoreLastra_A_B;		// Coordinata X punto interno n-esima lastra depositata  (CAVALLINA-CASSA)
	YInternoLastra_A_B : POINTER TO ARRAY [1..MAXFORMINGSLAB] OF ES_SpesoreLastra_A_B;		// Coordinata Y punto interno n-esima lastra depositata  (CAVALLINA-CASSA)
	ZInternoLastra_A_B : POINTER TO ARRAY [1..MAXFORMINGSLAB] OF ES_SpesoreLastra_A_B;		// Coordinata Z punto interno n-esima lastra depositata  (CAVALLINA-CASSA)
	XCentroLastra_A_B  : POINTER TO ARRAY [1..MAXFORMINGSLAB] OF ES_SpesoreLastra_A_B;		// Coordinata X punto centrale n-esima lastra depositata  (CAVALLINA-CASSA)
	YCentroLastra_A_B  : POINTER TO ARRAY [1..MAXFORMINGSLAB] OF ES_SpesoreLastra_A_B;		// Coordinata Y punto centrale n-esima lastra depositata  (CAVALLINA-CASSA)
	ZCentroLastra_A_B  : POINTER TO ARRAY [1..MAXFORMINGSLAB] OF ES_SpesoreLastra_A_B;		// Coordinata Z punto centrale n-esima lastra depositata  (CAVALLINA-CASSA)
	XEsternoLastra_A_B : POINTER TO ARRAY [1..MAXFORMINGSLAB] OF ES_SpesoreLastra_A_B;		// Coordinata X punto esterno n-esima lastra depositata  (CAVALLINA-CASSA)
	YEsternoLastra_A_B : POINTER TO ARRAY [1..MAXFORMINGSLAB] OF ES_SpesoreLastra_A_B;		// Coordinata Y punto esterno n-esima lastra depositata  (CAVALLINA-CASSA)
	ZEsternoLastra_A_B : POINTER TO ARRAY [1..MAXFORMINGSLAB] OF ES_SpesoreLastra_A_B;		
	
	YCoordinataAppoggioLastra_A_B : POINTER TO ARRAY [1..MAXFORMINGSLAB/2] OF ES_SpesoreLastra_A_B;
	ZCoordinataAppoggioLastra_A_B : POINTER TO ARRAY [1..MAXFORMINGSLAB/2] OF ES_SpesoreLastra_A_B;
	
	
	
END_VAR
VAR_OUTPUT
END_VAR
	
VAR
	Contador						: UINT;
	varEven							: UINT;
	LadoRegistarFor					: UINT;
	NuPieza_A						: UINT;
	NuPieza_B						: UINT;
	counter2						: INT;
END_VAR


CASE TipoCalForCavallete OF
{Region "Lato DX della cavallina "}
	
	1:	// Lato DX della cavallina
		FOR Contador := 1 TO numeroLastre_int * 2 DO 
			IF NOT 	CalculoEstacionPickinPiezasDiferentes THEN 
				varEven := Contador MOD 2;
					CASE varEven OF
						0:
							XFinale^[Contador] := Supporto^.XDim/2 + Supporto^.OFSDE_X180;
							CASE TipoRisultato OF 
								0:
									XFinale^[Contador] := Supporto^.XDim/2 + Supporto^.OFSDE_X180;
									ZFinale^[Contador] := ZInternoLastra^[(Contador+varEven)/2] + Supporto^.OFSDE_Z180;
								1:
									XFinale^[Contador] := Supporto^.XDim/2 + Supporto^.OFSDE_X180;
									ZFinale^[Contador] := ZInternoLastra^[(Contador+varEven)/2] + Supporto^.OFSDE_Z180;
								3:
									XFinale^[Contador] := Supporto^.XDim/2 + Supporto^.OFSDE_X180;
									ZFinale^[Contador] := ZInternoLastra^[(Contador+varEven)/2] + Supporto^.OFSDE_Z180;
								4:
									XFinale^[Contador] := Supporto^.XDim/2 + Supporto^.OFSDE_X180;
									ZFinale^[Contador] := ZInternoLastra^[(Contador+varEven)/2] + Supporto^.OFSDE_Z180;
							END_CASE
							JFinale^[Contador] := 180 - AlgoloAlfa_gradi + Supporto^.OFSDE_J180; 
						1: 
							XFinale^[Contador] := Supporto^.XDim/2 + Supporto^.OFSDE_X0;
							CASE TipoRisultato OF 
								1:	
										
										YFinale^[Contador] := YInternoLastra^[(Contador + varEven)/2] + Supporto^.OFSDE_Y0;
										ZFinale^[Contador] := ZInternoLastra^[(Contador+varEven)/2] 	+ Supporto^.OFSDE_Z0;
									2:	
										YFinale^[Contador] := YCentroLastra^[(Contador + varEven)/2] + Supporto^.OFSDE_Y0;
										ZFinale^[Contador] := ZCentroLastra^[(Contador + varEven)/2] + Supporto^.OFSDE_Z0;
									3:	
										YFinale^[Contador] := YEsternoLastra^[(Contador + varEven)/2] + Supporto^.OFSDE_Y0;
										ZFinale^[Contador] := ZEsternoLastra^[(Contador + varEven)/2] + Supporto^.OFSDE_Z0;
									4:	
										YFinale^[Contador] := YCoordinataAppoggioLastra^[(Contador + varEven)/2] + Supporto^.OFSDE_Y0;
										ZFinale^[Contador] := ZEsternoLastra^[(Contador + varEven)/2] + Supporto^.OFSDE_Z0;
								
							END_CASE
							 JFinale^[Contador] := AlgoloAlfa_gradi + Supporto^.OFSDE_J0;
					END_CASE
			ELSIF CalculoEstacionPickinPiezasDiferentes AND Supporto^.Tipologia = CAVALLETTO THEN 
				Fun_PiezaLadoCaballete(Nu_PiezaGlobal:= Contador , Grados:= ADR(LadoRegistarFor)  ,
										 Nu_pieza_LadoA=>NuPieza_A , Nu_pieza_LadoB=> NuPieza_B  );
				CASE TipoRisultato OF 
									1:	
										CASE LadoRegistarFor OF
											0: 
												CoorFinaleLado_Pri0_Des180^[NuPieza_A].LadoA.CoordenadaFinale_X := Supporto^.XDim/2 + Supporto^.OFSDE_X0;;
												CoorFinaleLado_Pri0_Des180^[NuPieza_A].LadoA.CoordenadaFinale_Y := YInternoLastra_A_B^[NuPieza_A].Lado_A_0Grados + Supporto^.OFSDE_Y0;
												CoorFinaleLado_Pri0_Des180^[NuPieza_A].LadoA.CoordenadaFinale_Z := ZInternoLastra_A_B^[NuPieza_A].Lado_A_0Grados + Supporto^.OFSDE_Z0;
												CoorFinaleLado_Pri0_Des180^[NuPieza_A].LadoA.CoordenadaFinale_J := AlgoloAlfa_gradi + Supporto^.OFSDE_J0 ;
											180 :
												 
												CoorFinaleLado_Pri0_Des180^[NuPieza_B].LadoB.CoordenadaFinale_X := Supporto^.XDim/2 + Supporto^.OFSDE_X180;;
												CoorFinaleLado_Pri0_Des180^[NuPieza_B].LadoB.CoordenadaFinale_Y := YInternoLastra_A_B^[NuPieza_B].Lado_B_180Grados + Supporto^.OFSDE_Y0;
												CoorFinaleLado_Pri0_Des180^[NuPieza_B].LadoB.CoordenadaFinale_Z := ZInternoLastra_A_B^[NuPieza_B].Lado_B_180Grados + Supporto^.OFSDE_Z0;
												CoorFinaleLado_Pri0_Des180^[NuPieza_B].LadoB.CoordenadaFinale_J := AlgoloAlfa_gradi + Supporto^.OFSDE_J0 ;
										END_CASE
									2:	
										CASE LadoRegistarFor OF
											0: 
												CoorFinaleLado_Pri0_Des180^[NuPieza_A].LadoA.CoordenadaFinale_X := Supporto^.XDim/2 + Supporto^.OFSDE_X0;;
												CoorFinaleLado_Pri0_Des180^[NuPieza_A].LadoA.CoordenadaFinale_Y := YCentroLastra_A_B^[NuPieza_A].Lado_A_0Grados + Supporto^.OFSDE_Y0;
												CoorFinaleLado_Pri0_Des180^[NuPieza_A].LadoA.CoordenadaFinale_Z := ZCentroLastra_A_B^[NuPieza_A].Lado_A_0Grados + Supporto^.OFSDE_Z0;
												CoorFinaleLado_Pri0_Des180^[NuPieza_A].LadoA.CoordenadaFinale_J := AlgoloAlfa_gradi + Supporto^.OFSDE_J0 ;
											180 :
												 
												CoorFinaleLado_Pri0_Des180^[NuPieza_B].LadoB.CoordenadaFinale_X := Supporto^.XDim/2 + Supporto^.OFSDE_X180;;
												CoorFinaleLado_Pri0_Des180^[NuPieza_B].LadoB.CoordenadaFinale_Y := YCentroLastra_A_B^[NuPieza_B].Lado_B_180Grados + Supporto^.OFSDE_Y0;
												CoorFinaleLado_Pri0_Des180^[NuPieza_B].LadoB.CoordenadaFinale_Z := ZCentroLastra_A_B^[NuPieza_B].Lado_B_180Grados + Supporto^.OFSDE_Z0;
												CoorFinaleLado_Pri0_Des180^[NuPieza_B].LadoB.CoordenadaFinale_J := AlgoloAlfa_gradi + Supporto^.OFSDE_J0 ;
										END_CASE
									3:	
										CASE LadoRegistarFor OF
											0: 
												CoorFinaleLado_Pri0_Des180^[NuPieza_A].LadoA.CoordenadaFinale_X := Supporto^.XDim/2 + Supporto^.OFSDE_X0;;
												CoorFinaleLado_Pri0_Des180^[NuPieza_A].LadoA.CoordenadaFinale_Y := YEsternoLastra_A_B^[NuPieza_A].Lado_A_0Grados + Supporto^.OFSDE_Y0;
												CoorFinaleLado_Pri0_Des180^[NuPieza_A].LadoA.CoordenadaFinale_Z := ZEsternoLastra_A_B^[NuPieza_A].Lado_A_0Grados + Supporto^.OFSDE_Z0;
												CoorFinaleLado_Pri0_Des180^[NuPieza_A].LadoA.CoordenadaFinale_J := AlgoloAlfa_gradi + Supporto^.OFSDE_J0 ;
											180 :
												 
												CoorFinaleLado_Pri0_Des180^[NuPieza_B].LadoB.CoordenadaFinale_X := Supporto^.XDim/2 + Supporto^.OFSDE_X180;;
												CoorFinaleLado_Pri0_Des180^[NuPieza_B].LadoB.CoordenadaFinale_Y := YEsternoLastra_A_B^[NuPieza_B].Lado_B_180Grados + Supporto^.OFSDE_Y0;
												CoorFinaleLado_Pri0_Des180^[NuPieza_B].LadoB.CoordenadaFinale_Z := ZEsternoLastra_A_B^[NuPieza_B].Lado_B_180Grados + Supporto^.OFSDE_Z0;
												CoorFinaleLado_Pri0_Des180^[NuPieza_B].LadoB.CoordenadaFinale_J := AlgoloAlfa_gradi + Supporto^.OFSDE_J0 ;
										END_CASE
									4:	
										CASE LadoRegistarFor OF
											0: 
												CoorFinaleLado_Pri0_Des180^[NuPieza_A].LadoA.CoordenadaFinale_X := Supporto^.XDim/2 + Supporto^.OFSDE_X0;;
												CoorFinaleLado_Pri0_Des180^[NuPieza_A].LadoA.CoordenadaFinale_Y := YCoordinataAppoggioLastra_A_B^[NuPieza_A].Lado_A_0Grados + Supporto^.OFSDE_Y0;
												CoorFinaleLado_Pri0_Des180^[NuPieza_A].LadoA.CoordenadaFinale_Z := ZCoordinataAppoggioLastra_A_B^[NuPieza_A].Lado_A_0Grados + Supporto^.OFSDE_Z0;
												CoorFinaleLado_Pri0_Des180^[NuPieza_A].LadoA.CoordenadaFinale_J := AlgoloAlfa_gradi + Supporto^.OFSDE_J0 ;
											180 :
												 
												CoorFinaleLado_Pri0_Des180^[NuPieza_B].LadoB.CoordenadaFinale_X := Supporto^.XDim/2 + Supporto^.OFSDE_X180;;
												CoorFinaleLado_Pri0_Des180^[NuPieza_B].LadoB.CoordenadaFinale_Y := YCoordinataAppoggioLastra_A_B^[NuPieza_B].Lado_B_180Grados + Supporto^.OFSDE_Y0;
												CoorFinaleLado_Pri0_Des180^[NuPieza_B].LadoB.CoordenadaFinale_Z := ZCoordinataAppoggioLastra_A_B^[NuPieza_B].Lado_B_180Grados + Supporto^.OFSDE_Z0;
												CoorFinaleLado_Pri0_Des180^[NuPieza_B].LadoB.CoordenadaFinale_J := AlgoloAlfa_gradi + Supporto^.OFSDE_J0 ;
										END_CASE
																		
					END_CASE
							
			END_IF

	END_FOR 
{endregion}

{Region "Ordinamento consecutivo prima un lato poi l'altro"}


		(* Ordinamento consecutivo prima un lato poi l'altro *)
		2:
			FOR Contador :=1 TO numeroLastre_int BY 1 DO
				Fun_PiezaLadoCaballete(Nu_PiezaGlobal:= Contador , Grados:= ADR(LadoRegistarFor)  ,
										 Nu_pieza_LadoA=>NuPieza_A , Nu_pieza_LadoB=> NuPieza_B  );
				IF NOT CalculoEstacionPickinPiezasDiferentes THEN 
					CASE TipoRisultato OF 
							1:	
								
								CoorFinaleLado_Pri0_Des180^[Contador].LadoA.CoordenadaFinale_Y := YInternoLastra^[Contador] + Supporto^.OFSDE_Y0;
								CoorFinaleLado_Pri0_Des180^[Contador].LadoA.CoordenadaFinale_Z := ZInternoLastra^[Contador] + Supporto^.OFSDE_Z0;
								
								CoorFinaleLado_Pri0_Des180^[Contador].LadoB.CoordenadaFinale_Y := -YInternoLastra^[Contador] + Supporto^.OFSDE_Y180;
								CoorFinaleLado_Pri0_Des180^[Contador].LadoB.CoordenadaFinale_Z := ZInternoLastra^[Contador] + Supporto^.OFSDE_Z180;
								
									
	
							2:
								CoorFinaleLado_Pri0_Des180^[Contador].LadoA.CoordenadaFinale_Y := YCentroLastra^[Contador] + Supporto^.OFSDE_Y0;
								CoorFinaleLado_Pri0_Des180^[Contador].LadoA.CoordenadaFinale_Z := ZCentroLastra^[Contador] + Supporto^.OFSDE_Z0;
								
								CoorFinaleLado_Pri0_Des180^[Contador].LadoB.CoordenadaFinale_Y := -YCentroLastra^[Contador] + Supporto^.OFSDE_Y180;
								CoorFinaleLado_Pri0_Des180^[Contador].LadoB.CoordenadaFinale_Z := ZCentroLastra^[Contador] + Supporto^.OFSDE_Z180;
							
							3:
								CoorFinaleLado_Pri0_Des180^[Contador].LadoA.CoordenadaFinale_Y := YEsternoLastra^[Contador] + Supporto^.OFSDE_Y0;
								CoorFinaleLado_Pri0_Des180^[Contador].LadoA.CoordenadaFinale_Z := ZEsternoLastra^[Contador] + Supporto^.OFSDE_Z0;
								
								CoorFinaleLado_Pri0_Des180^[Contador].LadoB.CoordenadaFinale_Y := -YEsternoLastra^[Contador] + Supporto^.OFSDE_Y180;
								CoorFinaleLado_Pri0_Des180^[Contador].LadoB.CoordenadaFinale_Z := ZEsternoLastra^[Contador] + Supporto^.OFSDE_Z180;
							
							4:
								CoorFinaleLado_Pri0_Des180^[Contador].LadoA.CoordenadaFinale_Y := YCoordinataAppoggioLastra^[Contador] + Supporto^.OFSDE_Y0;
								CoorFinaleLado_Pri0_Des180^[Contador].LadoA.CoordenadaFinale_Z := ZEsternoLastra^[Contador] + Supporto^.OFSDE_Z0;
								
								CoorFinaleLado_Pri0_Des180^[Contador].LadoB.CoordenadaFinale_Y := -YCoordinataAppoggioLastra^[Contador] + Supporto^.OFSDE_Y180;
								CoorFinaleLado_Pri0_Des180^[Contador].LadoB.CoordenadaFinale_Z := ZEsternoLastra^[Contador] + Supporto^.OFSDE_Z180;
	
					END_CASE
					CoorFinaleLado_Pri0_Des180^[Contador].LadoA.CoordenadaFinale_X := Supporto^.XDim/2 + Supporto^.OFSDE_X180;
					CoorFinaleLado_Pri0_Des180^[Contador].LadoA.CoordenadaFinale_J :=  AlgoloAlfa_gradi + Supporto^.OFSDE_J0;
					CoorFinaleLado_Pri0_Des180^[Contador].LadoB.CoordenadaFinale_J := 180 - AlgoloAlfa_gradi + Supporto^.OFSDE_J180;
				ELSIF  CalculoEstacionPickinPiezasDiferentes AND Supporto^.Tipologia = CAVALLETTO  THEN 	
					
					CASE TipoRisultato OF
						1:
							CASE LadoRegistarFor OF
								0:
									CoorFinaleLado_Pri0_Des180^[NuPieza_A].LadoA.CoordenadaFinale_X := Supporto^.XDim/2 + Supporto^.OFSDE_X180;
									CoorFinaleLado_Pri0_Des180^[NuPieza_A].LadoA.CoordenadaFinale_Y := YInternoLastra_A_B^[NuPieza_A].Lado_A_0Grados + Supporto^.OFSDE_Y0;
									CoorFinaleLado_Pri0_Des180^[NuPieza_A].LadoA.CoordenadaFinale_Z := ZInternoLastra_A_B^[NuPieza_A].Lado_A_0Grados + Supporto^.OFSDE_Z0;
									CoorFinaleLado_Pri0_Des180^[NuPieza_A].LadoA.CoordenadaFinale_J := AlgoloAlfa_gradi + Supporto^.OFSDE_J0;
									
								180:
									CoorFinaleLado_Pri0_Des180^[NuPieza_B].LadoA.CoordenadaFinale_X := Supporto^.XDim/2 + Supporto^.OFSDE_X180;
									CoorFinaleLado_Pri0_Des180^[NuPieza_B].LadoB.CoordenadaFinale_Y := -YInternoLastra_A_B^[NuPieza_B].Lado_B_180Grados + Supporto^.OFSDE_Y180;
									CoorFinaleLado_Pri0_Des180^[NuPieza_B].LadoB.CoordenadaFinale_Z := ZInternoLastra_A_B^[NuPieza_B].Lado_B_180Grados + Supporto^.OFSDE_Z180;
									CoorFinaleLado_Pri0_Des180^[NuPieza_B].LadoB.CoordenadaFinale_J := 180 - AlgoloAlfa_gradi + Supporto^.OFSDE_J180;
							END_CASE
						
						
						2:
							CASE LadoRegistarFor OF
								0:
									CoorFinaleLado_Pri0_Des180^[NuPieza_A].LadoA.CoordenadaFinale_X := Supporto^.XDim/2 + Supporto^.OFSDE_X180;
									CoorFinaleLado_Pri0_Des180^[NuPieza_A].LadoA.CoordenadaFinale_Y := YCentroLastra_A_B^[NuPieza_A].Lado_A_0Grados + Supporto^.OFSDE_Y0;
									CoorFinaleLado_Pri0_Des180^[NuPieza_A].LadoA.CoordenadaFinale_Z := ZCentroLastra_A_B^[NuPieza_A].Lado_A_0Grados + Supporto^.OFSDE_Z0;
									CoorFinaleLado_Pri0_Des180^[NuPieza_A].LadoA.CoordenadaFinale_J := AlgoloAlfa_gradi + Supporto^.OFSDE_J0;
								180:
									CoorFinaleLado_Pri0_Des180^[NuPieza_B].LadoA.CoordenadaFinale_X := Supporto^.XDim/2 + Supporto^.OFSDE_X180;
									CoorFinaleLado_Pri0_Des180^[NuPieza_B].LadoB.CoordenadaFinale_Y := -YCentroLastra_A_B^[NuPieza_B].Lado_B_180Grados + Supporto^.OFSDE_Y180;
									CoorFinaleLado_Pri0_Des180^[NuPieza_B].LadoB.CoordenadaFinale_Z := ZCentroLastra_A_B^[NuPieza_B].Lado_B_180Grados + Supporto^.OFSDE_Z180;
									CoorFinaleLado_Pri0_Des180^[NuPieza_B].LadoB.CoordenadaFinale_J := 180 - AlgoloAlfa_gradi + Supporto^.OFSDE_J180;
							END_CASE
						3:
							CASE LadoRegistarFor OF
								0:
									CoorFinaleLado_Pri0_Des180^[NuPieza_A].LadoA.CoordenadaFinale_X := Supporto^.XDim/2 + Supporto^.OFSDE_X180;
									CoorFinaleLado_Pri0_Des180^[NuPieza_A].LadoA.CoordenadaFinale_Y := YEsternoLastra_A_B^[NuPieza_A].Lado_A_0Grados + Supporto^.OFSDE_Y0;
									CoorFinaleLado_Pri0_Des180^[NuPieza_A].LadoA.CoordenadaFinale_Z := ZEsternoLastra_A_B^[NuPieza_A].Lado_A_0Grados + Supporto^.OFSDE_Z0;
									CoorFinaleLado_Pri0_Des180^[NuPieza_A].LadoA.CoordenadaFinale_J := AlgoloAlfa_gradi + Supporto^.OFSDE_J0;
								180:
									CoorFinaleLado_Pri0_Des180^[NuPieza_B].LadoA.CoordenadaFinale_X := Supporto^.XDim/2 + Supporto^.OFSDE_X180;
									CoorFinaleLado_Pri0_Des180^[NuPieza_B].LadoB.CoordenadaFinale_Y := -YEsternoLastra_A_B^[NuPieza_B].Lado_B_180Grados + Supporto^.OFSDE_Y180;
									CoorFinaleLado_Pri0_Des180^[NuPieza_B].LadoB.CoordenadaFinale_Z := ZEsternoLastra_A_B^[NuPieza_B].Lado_B_180Grados + Supporto^.OFSDE_Z180;
									CoorFinaleLado_Pri0_Des180^[NuPieza_B].LadoB.CoordenadaFinale_J := 180 - AlgoloAlfa_gradi + Supporto^.OFSDE_J180;
							END_CASE
						4:
							CASE LadoRegistarFor OF
								0:
									CoorFinaleLado_Pri0_Des180^[NuPieza_A].LadoA.CoordenadaFinale_X := Supporto^.XDim/2 + Supporto^.OFSDE_X180;
									CoorFinaleLado_Pri0_Des180^[NuPieza_A].LadoA.CoordenadaFinale_Y := YCoordinataAppoggioLastra_A_B^[NuPieza_A].Lado_A_0Grados + Supporto^.OFSDE_Y0;
									CoorFinaleLado_Pri0_Des180^[NuPieza_A].LadoA.CoordenadaFinale_Z := ZEsternoLastra_A_B^[NuPieza_A].Lado_A_0Grados + Supporto^.OFSDE_Z0;
									CoorFinaleLado_Pri0_Des180^[NuPieza_A].LadoA.CoordenadaFinale_J := AlgoloAlfa_gradi + Supporto^.OFSDE_J0;
								180:
									CoorFinaleLado_Pri0_Des180^[NuPieza_B].LadoA.CoordenadaFinale_X := Supporto^.XDim/2 + Supporto^.OFSDE_X180;
									CoorFinaleLado_Pri0_Des180^[NuPieza_B].LadoB.CoordenadaFinale_Y := -YCoordinataAppoggioLastra_A_B^[NuPieza_B].Lado_B_180Grados + Supporto^.OFSDE_Y180;
									CoorFinaleLado_Pri0_Des180^[NuPieza_B].LadoB.CoordenadaFinale_Z := ZEsternoLastra_A_B^[NuPieza_B].Lado_B_180Grados + Supporto^.OFSDE_Z180;
									CoorFinaleLado_Pri0_Des180^[NuPieza_B].LadoB.CoordenadaFinale_J := 180 - AlgoloAlfa_gradi + Supporto^.OFSDE_J180;
							END_CASE
						
						
						
						
						
					END_CASE
				
				END_IF
				
				
				
				
				
				
			END_FOR
		













{endregion}
END_CASE

END_FUNCTION_BLOCK

// ---- Data types/AlbertoPruevas/BloqueFunciones/CalculoFormaciones/Fb_Fb_CalculoTodo0CoordenadasFinales.TcPOU
FUNCTION_BLOCK Fb_Fb_CalculoTodo0CoordenadasFinales
VAR_INPUT
	CalculoEstacionPickinPiezasDiferentes		: BOOL;
	numeroLastre_int			:UINT;
	TipoCalForCavallete  					:UINT ;
	TipoRisultato				:UINT;
	AlgoloAlfa_gradi			:LREAL;
	
	Supporto :POINTER TO  TFMachinePalletizer_Pallet;
	
	YCoordinataAppoggioLastra :POINTER TO  ARRAY [1..MAXFORMINGSLAB/2] OF LREAL;		// Coordinata Y del punto di appoggio della lastra sulla base della cavallina  (CAVALLINA-INCLINATO)
	ZCoordinataAppoggioLastra :POINTER TO  ARRAY [1..MAXFORMINGSLAB/2] OF LREAL;		// Coordinata Z del punto di appoggio della lastra sulla base della cavallina  (CAVALLINA-INCLINATO)
	
	YCoordinataAppoggioLastra_A_B :POINTER TO  ARRAY [1..MAXFORMINGSLAB/2] OF ES_SpesoreLastra_A_B;
	ZCoordinataAppoggioLastra_A_B :POINTER TO  ARRAY [1..MAXFORMINGSLAB/2] OF ES_SpesoreLastra_A_B;
	
	XFinaleLado_0Grados :POINTER TO ARRAY [1..MAXFORMINGSLAB] OF LREAL;		// Coordinata X punto finale n-esima lastra/falda depositata
	YFinaleLado_0Grados :POINTER TO ARRAY [1..MAXFORMINGSLAB] OF LREAL;		// Coordinata Y punto finale n-esima lastra/falda depositata
	ZFinaleLado_0Grados :POINTER TO ARRAY [1..MAXFORMINGSLAB] OF LREAL;		// Coordinata Z punto finale n-esima lastra/falda depositata
	JFinaleLado_0Grados :POINTER TO ARRAY [1..MAXFORMINGSLAB] OF LREAL;		// Coordinata J punto finale n-esima lastra/falda depositata
	
	XInternoLastra :POINTER TO  ARRAY [1..MAXFORMINGSLAB] OF LREAL;		// Coordinata X punto interno n-esima lastra depositata  (CAVALLINA-CASSA)
	YInternoLastra :POINTER TO  ARRAY [1..MAXFORMINGSLAB] OF LREAL;		// Coordinata Y punto interno n-esima lastra depositata  (CAVALLINA-CASSA)
	ZInternoLastra :POINTER TO  ARRAY [1..MAXFORMINGSLAB] OF LREAL;		// Coordinata Z punto interno n-esima lastra depositata  (CAVALLINA-CASSA)
	XCentroLastra  :POINTER TO  ARRAY [1..MAXFORMINGSLAB] OF LREAL;		// Coordinata X punto centrale n-esima lastra depositata  (CAVALLINA-CASSA)
	YCentroLastra  :POINTER TO  ARRAY [1..MAXFORMINGSLAB] OF LREAL;		// Coordinata Y punto centrale n-esima lastra depositata  (CAVALLINA-CASSA)
	ZCentroLastra  :POINTER TO  ARRAY [1..MAXFORMINGSLAB] OF LREAL;		// Coordinata Z punto centrale n-esima lastra depositata  (CAVALLINA-CASSA)
	XEsternoLastra :POINTER TO  ARRAY [1..MAXFORMINGSLAB] OF LREAL;		// Coordinata X punto esterno n-esima lastra depositata  (CAVALLINA-CASSA)
	YEsternoLastra :POINTER TO  ARRAY [1..MAXFORMINGSLAB] OF LREAL;		// Coordinata Y punto esterno n-esima lastra depositata  (CAVALLINA-CASSA)
	ZEsternoLastra :POINTER TO  ARRAY [1..MAXFORMINGSLAB] OF LREAL;		// Coordinata Z punto esterno n-esima lastra depositata  (CAVALLINA-CASSA)
	
	XInternoLastra_A_B :POINTER TO ARRAY [1..MAXFORMINGSLAB] OF ES_SpesoreLastra_A_B;		// Coordinata X punto interno n-esima lastra depositata  (CAVALLINA-CASSA)
	YInternoLastra_A_B :POINTER TO ARRAY [1..MAXFORMINGSLAB] OF ES_SpesoreLastra_A_B;		// Coordinata Y punto interno n-esima lastra depositata  (CAVALLINA-CASSA)
	ZInternoLastra_A_B :POINTER TO ARRAY [1..MAXFORMINGSLAB] OF ES_SpesoreLastra_A_B;		// Coordinata Z punto interno n-esima lastra depositata  (CAVALLINA-CASSA)
	XCentroLastra_A_B  :POINTER TO ARRAY [1..MAXFORMINGSLAB] OF ES_SpesoreLastra_A_B;		// Coordinata X punto centrale n-esima lastra depositata  (CAVALLINA-CASSA)
	YCentroLastra_A_B  :POINTER TO ARRAY [1..MAXFORMINGSLAB] OF ES_SpesoreLastra_A_B;		// Coordinata Y punto centrale n-esima lastra depositata  (CAVALLINA-CASSA)
	ZCentroLastra_A_B  :POINTER TO ARRAY [1..MAXFORMINGSLAB] OF ES_SpesoreLastra_A_B;		// Coordinata Z punto centrale n-esima lastra depositata  (CAVALLINA-CASSA)
	XEsternoLastra_A_B :POINTER TO ARRAY [1..MAXFORMINGSLAB] OF ES_SpesoreLastra_A_B;		// Coordinata X punto esterno n-esima lastra depositata  (CAVALLINA-CASSA)
	YEsternoLastra_A_B :POINTER TO ARRAY [1..MAXFORMINGSLAB] OF ES_SpesoreLastra_A_B;		// Coordinata Y punto esterno n-esima lastra depositata  (CAVALLINA-CASSA)
	ZEsternoLastra_A_B :POINTER TO ARRAY [1..MAXFORMINGSLAB] OF ES_SpesoreLastra_A_B;		// Coordinata Z punto esterno n-esima lastra depositata  (CAVALLINA-CASSA)
END_VAR
VAR_OUTPUT
END_VAR
VAR
	Contador: INT;
END_VAR


IF TipoCalForCavallete = 3 THEN 
	
		FOR Contador:=1 TO numeroLastre_int BY 1 DO
						
			XFinaleLado_0Grados^[Contador] := Supporto^.XDim/2 + Supporto^.OFSDE_X0;
			
				IF  NOT CalculoEstacionPickinPiezasDiferentes	THEN	
					CASE TipoRisultato OF
						1:	
							YFinaleLado_0Grados^[Contador] := YInternoLastra^[Contador] + Supporto^.OFSDE_Y0;
							ZFinaleLado_0Grados^[Contador] := ZInternoLastra^[Contador] + Supporto^.OFSDE_Z0;
							
						2:	
							YFinaleLado_0Grados^[Contador] := YCentroLastra^[Contador] + Supporto^.OFSDE_Y0;
							ZFinaleLado_0Grados^[Contador] := ZCentroLastra^[Contador] + Supporto^.OFSDE_Z0;
						3:	
							YFinaleLado_0Grados^[Contador] := YEsternoLastra^[Contador] + Supporto^.OFSDE_Y0;
							ZFinaleLado_0Grados^[Contador] := ZEsternoLastra^[Contador] + Supporto^.OFSDE_Z0;
						4:	
							YFinaleLado_0Grados^[Contador] := YCoordinataAppoggioLastra^[Contador] + Supporto^.OFSDE_Y0;
							ZFinaleLado_0Grados^[Contador] := ZEsternoLastra^[Contador] + Supporto^.OFSDE_Z0;
					END_CASE
				ELSIF CalculoEstacionPickinPiezasDiferentes	THEN
					CASE TipoRisultato OF
						1:	
							YFinaleLado_0Grados^[Contador] := YInternoLastra_A_B^[Contador].Lado_A_0Grados + Supporto^.OFSDE_Y0;
							ZFinaleLado_0Grados^[Contador] := ZInternoLastra_A_B^[Contador].Lado_A_0Grados + Supporto^.OFSDE_Z0;	
							
						2:	
							
							YFinaleLado_0Grados^[Contador] := YCentroLastra_A_B^[Contador].Lado_A_0Grados + Supporto^.OFSDE_Y0;
							ZFinaleLado_0Grados^[Contador] := ZCentroLastra_A_B^[Contador].Lado_A_0Grados + Supporto^.OFSDE_Z0;
						3:	
							YFinaleLado_0Grados^[Contador] := YEsternoLastra_A_B^[Contador].Lado_A_0Grados + Supporto^.OFSDE_Y0;
							ZFinaleLado_0Grados^[Contador] := ZEsternoLastra_A_B^[Contador].Lado_A_0Grados + Supporto^.OFSDE_Z0;
						4:	
							YFinaleLado_0Grados^[Contador] := YCoordinataAppoggioLastra_A_B^[Contador].Lado_A_0Grados + Supporto^.OFSDE_Y0;
							ZFinaleLado_0Grados^[Contador] := ZEsternoLastra_A_B^[Contador].Lado_A_0Grados + Supporto^.OFSDE_Z0;
					END_CASE
				END_IF
			
			JFinaleLado_0Grados^[Contador] := AlgoloAlfa_gradi + Supporto^.OFSDE_J0;
		END_FOR
END_IF

END_FUNCTION_BLOCK

// ---- Data types/AlbertoPruevas/BloqueFunciones/CalculoFormaciones/Fb_CalculoTodo180CoordenadasFinales.TcPOU
FUNCTION_BLOCK Fb_CalculoTodo180CoordenadasFinales
VAR_INPUT
	CalculoEstacionPickinPiezasDiferentes		: BOOL;
	numeroLastre_int			:UINT;
	TipoCalForCavallete  					:UINT ;
	TipoRisultato				:UINT;
	AlgoloAlfa_gradi			: LREAL;
	
	Supporto :POINTER TO  TFMachinePalletizer_Pallet;
	
	YCoordinataAppoggioLastra :POINTER TO  ARRAY [1..MAXFORMINGSLAB/2] OF LREAL;		// Coordinata Y del punto di appoggio della lastra sulla base della cavallina  (CAVALLINA-INCLINATO)
	ZCoordinataAppoggioLastra :POINTER TO  ARRAY [1..MAXFORMINGSLAB/2] OF LREAL;		// Coordinata Z del punto di appoggio della lastra sulla base della cavallina  (CAVALLINA-INCLINATO)
	
	YCoordinataAppoggioLastra_A_B :POINTER TO  ARRAY [1..MAXFORMINGSLAB/2] OF ES_SpesoreLastra_A_B;
	ZCoordinataAppoggioLastra_A_B :POINTER TO  ARRAY [1..MAXFORMINGSLAB/2] OF ES_SpesoreLastra_A_B;
	
	XFinaleLado_180Grados :POINTER TO ARRAY [1..MAXFORMINGSLAB] OF LREAL;		// Coordinata X punto finale n-esima lastra/falda depositata
	YFinaleLado_180Grados :POINTER TO ARRAY [1..MAXFORMINGSLAB] OF LREAL;		// Coordinata Y punto finale n-esima lastra/falda depositata
	ZFinaleLado_180Grados :POINTER TO ARRAY [1..MAXFORMINGSLAB] OF LREAL;		// Coordinata Z punto finale n-esima lastra/falda depositata
	JFinaleLado_180Grados :POINTER TO ARRAY [1..MAXFORMINGSLAB] OF LREAL;		// Coordinata J punto finale n-esima lastra/falda depositata
	
	XInternoLastra :POINTER TO  ARRAY [1..MAXFORMINGSLAB] OF LREAL;		// Coordinata X punto interno n-esima lastra depositata  (CAVALLINA-CASSA)
	YInternoLastra :POINTER TO  ARRAY [1..MAXFORMINGSLAB] OF LREAL;		// Coordinata Y punto interno n-esima lastra depositata  (CAVALLINA-CASSA)
	ZInternoLastra :POINTER TO  ARRAY [1..MAXFORMINGSLAB] OF LREAL;		// Coordinata Z punto interno n-esima lastra depositata  (CAVALLINA-CASSA)
	XCentroLastra  :POINTER TO  ARRAY [1..MAXFORMINGSLAB] OF LREAL;		// Coordinata X punto centrale n-esima lastra depositata  (CAVALLINA-CASSA)
	YCentroLastra  :POINTER TO  ARRAY [1..MAXFORMINGSLAB] OF LREAL;		// Coordinata Y punto centrale n-esima lastra depositata  (CAVALLINA-CASSA)
	ZCentroLastra  :POINTER TO  ARRAY [1..MAXFORMINGSLAB] OF LREAL;		// Coordinata Z punto centrale n-esima lastra depositata  (CAVALLINA-CASSA)
	XEsternoLastra :POINTER TO  ARRAY [1..MAXFORMINGSLAB] OF LREAL;		// Coordinata X punto esterno n-esima lastra depositata  (CAVALLINA-CASSA)
	YEsternoLastra :POINTER TO  ARRAY [1..MAXFORMINGSLAB] OF LREAL;		// Coordinata Y punto esterno n-esima lastra depositata  (CAVALLINA-CASSA)
	ZEsternoLastra :POINTER TO  ARRAY [1..MAXFORMINGSLAB] OF LREAL;		// Coordinata Z punto esterno n-esima lastra depositata  (CAVALLINA-CASSA)
	
	XInternoLastra_A_B :POINTER TO ARRAY [1..MAXFORMINGSLAB] OF ES_SpesoreLastra_A_B;		// Coordinata X punto interno n-esima lastra depositata  (CAVALLINA-CASSA)
	YInternoLastra_A_B :POINTER TO ARRAY [1..MAXFORMINGSLAB] OF ES_SpesoreLastra_A_B;		// Coordinata Y punto interno n-esima lastra depositata  (CAVALLINA-CASSA)
	ZInternoLastra_A_B :POINTER TO ARRAY [1..MAXFORMINGSLAB] OF ES_SpesoreLastra_A_B;		// Coordinata Z punto interno n-esima lastra depositata  (CAVALLINA-CASSA)
	XCentroLastra_A_B  :POINTER TO ARRAY [1..MAXFORMINGSLAB] OF ES_SpesoreLastra_A_B;		// Coordinata X punto centrale n-esima lastra depositata  (CAVALLINA-CASSA)
	YCentroLastra_A_B  :POINTER TO ARRAY [1..MAXFORMINGSLAB] OF ES_SpesoreLastra_A_B;		// Coordinata Y punto centrale n-esima lastra depositata  (CAVALLINA-CASSA)
	ZCentroLastra_A_B  :POINTER TO ARRAY [1..MAXFORMINGSLAB] OF ES_SpesoreLastra_A_B;		// Coordinata Z punto centrale n-esima lastra depositata  (CAVALLINA-CASSA)
	XEsternoLastra_A_B :POINTER TO ARRAY [1..MAXFORMINGSLAB] OF ES_SpesoreLastra_A_B;		// Coordinata X punto esterno n-esima lastra depositata  (CAVALLINA-CASSA)
	YEsternoLastra_A_B :POINTER TO ARRAY [1..MAXFORMINGSLAB] OF ES_SpesoreLastra_A_B;		// Coordinata Y punto esterno n-esima lastra depositata  (CAVALLINA-CASSA)
	ZEsternoLastra_A_B :POINTER TO ARRAY [1..MAXFORMINGSLAB] OF ES_SpesoreLastra_A_B;		// Coordinata Z punto esterno n-esima lastra depositata  (CAVALLINA-CASSA)
END_VAR

VAR_OUTPUT
END_VAR
VAR
	Contador: INT;
	
	
END_VAR

IF TipoCalForCavallete = 4 THEN 

		FOR Contador:=1 TO numeroLastre_int BY 1 DO
						
			XFinaleLado_180Grados^[Contador] := Supporto^.XDim/2 + Supporto^.OFSDE_X180;
			
				IF  NOT CalculoEstacionPickinPiezasDiferentes	THEN	
					CASE TipoRisultato OF
						1:	
							YFinaleLado_180Grados^[Contador] := -YInternoLastra^[Contador] + Supporto^.OFSDE_Y180;
							ZFinaleLado_180Grados^[Contador] := ZInternoLastra^[Contador] + Supporto^.OFSDE_Z180;
							
						2:	
							YFinaleLado_180Grados^[Contador] := -YCentroLastra^[Contador] + Supporto^.OFSDE_Y180;
							ZFinaleLado_180Grados^[Contador] := ZCentroLastra^[Contador] + Supporto^.OFSDE_Z180;
						3:	
							YFinaleLado_180Grados^[Contador] := -YEsternoLastra^[Contador] + Supporto^.OFSDE_Y180;
							ZFinaleLado_180Grados^[Contador] := ZEsternoLastra^[Contador] + Supporto^.OFSDE_Z180;
						4:	
							YFinaleLado_180Grados^[Contador] := -YCoordinataAppoggioLastra^[Contador] + Supporto^.OFSDE_Y180;
							ZFinaleLado_180Grados^[Contador] := ZEsternoLastra^[Contador] + Supporto^.OFSDE_Z180;
					END_CASE
				ELSIF CalculoEstacionPickinPiezasDiferentes	THEN
					CASE TipoRisultato OF
						1:	
							YFinaleLado_180Grados^[Contador] := -YInternoLastra_A_B^[Contador].Lado_B_180Grados + Supporto^.OFSDE_Y180;
							ZFinaleLado_180Grados^[Contador] := ZInternoLastra_A_B^[Contador].Lado_B_180Grados + Supporto^.OFSDE_Z180;	
							
						2:	
							
							YFinaleLado_180Grados^[Contador] := -YCentroLastra_A_B^[Contador].Lado_B_180Grados + Supporto^.OFSDE_Y180;
							ZFinaleLado_180Grados^[Contador] := ZCentroLastra_A_B^[Contador].Lado_B_180Grados + Supporto^.OFSDE_Z180;
						3:	
							YFinaleLado_180Grados^[Contador] := -YEsternoLastra_A_B^[Contador].Lado_B_180Grados + Supporto^.OFSDE_Y180;
							ZFinaleLado_180Grados^[Contador] := ZEsternoLastra_A_B^[Contador].Lado_B_180Grados + Supporto^.OFSDE_Z180;
						4:	
							YFinaleLado_180Grados^[Contador] := -YCoordinataAppoggioLastra_A_B^[Contador].Lado_B_180Grados + Supporto^.OFSDE_Y180;
							ZFinaleLado_180Grados^[Contador] := ZEsternoLastra_A_B^[Contador].Lado_B_180Grados + Supporto^.OFSDE_Z180;
					END_CASE
				END_IF
			
			JFinaleLado_180Grados^[Contador] := 180 - AlgoloAlfa_gradi + Supporto^.OFSDE_J180; 
		END_FOR
END_IF

END_FUNCTION_BLOCK

// ---- Data types/AlbertoPruevas/Funciones/Fun_NumeroPiezasLadoCaballete.TcPOU
FUNCTION Fun_NumeroPiezasLadoCaballete : bool
VAR_INPUT
	NuPieasTotales 	: UINT ;
	PiezasLadoA		: POINTER TO UINT ;
	PiezasLadoB		: POINTER TO UINT ;
END_VAR
VAR
END_VAR

IF (NuPieasTotales MOD 2 = 1) THEN 
	PiezasLadoA^ := ( NuPieasTotales / 2) + 1  ;
	PiezasLadoB^ := ( NuPieasTotales / 2)  ;
ELSE
	PiezasLadoA^ := ( NuPieasTotales / 2)   ;
	PiezasLadoB^ := ( NuPieasTotales / 2)  ;
END_IF

END_FUNCTION

// ---- POUs/TFPalletizerData_Lastre/TFGetEnableCode_Lastre.TcPOU
FUNCTION TFGetEnableCode_Lastre : ARRAY [1..MAXFORMINGCODE*MAXFORMING] OF INT
VAR_INPUT
	Forming : POINTER TO ARRAY [1..MAXFORMING] OF TFMachinePalletizer_FormingForSlab;
END_VAR
VAR
	EnableCode : ARRAY [1..MAXFORMINGCODE*MAXFORMING] OF INT;
	pp : UINT;
	pf : UINT;
	c : INT;
	i : UINT;
END_VAR

FOR i:=1 TO MAXFORMINGCODE*MAXFORMING DO
	EnableCode[i]:= 0;
END_FOR
c:=1; 
(* Per Tutte le Formature Attive *)
FOR pf:=1 TO MAXFORMING DO
	IF Forming^[pf].Enable = 1 THEN
		(* Per tutti i codici di Pallettizzazione Validi *)
		FOR pp:=1 TO MAXFORMINGCODE DO
			IF Forming^[pf].Code[pp] > 0 THEN
				EnableCode[c] := Forming^[pf].Code[pp];
				c := c+1;
			END_IF
		END_FOR
	END_IF
END_FOR
TFGetEnableCode_Lastre := EnableCode;

END_FUNCTION

// ---- POUs/TFPalletizerData_Lastre/TFWAM_RicavaListaInLavoro.TcPOU
(*Funzione che restituisce il numero della postazione avente una lista in lavorazione*)
FUNCTION TFWAM_RicavaListaInLavoro : UINT
VAR_INPUT
	WorkAreaProductionList : POINTER TO ARRAY [1..MAXAREA] OF TFMachinePalletizer_ListaProduzione_WAM; //Lista di produzione che devo Svolgere PER ogni POSTAZIONE
END_VAR
VAR
	i:UINT;
END_VAR

(* Ciclo tutte le Liste *)
FOR i:=1 TO MAXAREAPRESENT DO
	(* Se Lista NON è già stata avviata e NON è TERMINATA*)
	IF WorkAreaProductionList^[i].Stato >= LISTA_PROD_IN_ESECUZIONE AND WorkAreaProductionList^[i].Stato < LISTA_PROD_ESEGUITA THEN
		TFWAM_RicavaListaInLavoro := i;
		RETURN;
	END_IF
END_FOR
TFWAM_RicavaListaInLavoro:=0;

END_FUNCTION

// ---- POUs/TFPalletizerData_Lastre/TFPalletizer_CalcolaCoordinataPrelievo_PickPoint.TcPOU
FUNCTION TFPalletizer_CalcolaCoordinataPrelievo_PickPoint : LREAL
VAR_INPUT
	WorkPickPoint : POINTER TO ARRAY [1..MAXPICKPOINT] OF TFMachinePalletizer_WorkPickPointSlab;
	WorkPickPointState : POINTER TO ARRAY [1..MAXPICKPOINT] OF TFMachinePalletizer_WorkPickPoint_State;
	WorkPickPointOffset : POINTER TO ARRAY [1..MAXPICKPOINT] OF TFMachinePalletizer_WorkPickPointOffset;
	NPickPoint : UINT;			//Numero PickPoint del quale si vuole la coordinata
	AsseDaCalcolare : STRING;	//Nome dell'Asse del quale si vuole calcolare la coordinata 
END_VAR
VAR
	wpp : INT;
	Ncase : INT;
END_VAR

TFPalletizer_CalcolaCoordinataPrelievo_PickPoint := 0;
IF AsseDaCalcolare = 'X' THEN
	Ncase	:= 1;
ELSIF AsseDaCalcolare = 'Y' THEN
	Ncase	:= 2;
ELSIF AsseDaCalcolare = 'Z' THEN
	Ncase	:= 3;
ELSIF AsseDaCalcolare = 'J' THEN
	Ncase	:= 4;
END_IF

IF WorkPickPoint^[NPickPoint].Tipologia = WA_CON_PALLET  OR WorkPickPoint^[NPickPoint].Tipologia = WA_CON_CASSA OR WorkPickPoint^[NPickPoint].Tipologia = WA_CON_CAVALLINA THEN
	CASE Ncase OF
		1:
			TFPalletizer_CalcolaCoordinataPrelievo_PickPoint := WorkPickPoint^[NPickPoint].X +							// Quota X centro Rulliera	
																//WorkPickPointState^[NPickPoint].XPosBandella +	// Quota Relativa della posizione della bandella
																//(WorkPickPointState^[NPickPoint].Element.XDim/2) +		// Metà Lunghezza Lastra
																WorkPickPointOffset^[NPickPoint].X;						// Valore di Offset Di Prelievo in X	
		
		2:	
			TFPalletizer_CalcolaCoordinataPrelievo_PickPoint := WorkPickPoint^[NPickPoint].Y -							// Quota Y centro Rulliera	
																//WorkPickPointState^[NPickPoint].YPosBandella +	// Quota Relativa della posizione della bandella
																(WorkPickPointState^[NPickPoint].Element.YDim/2) +		// Metà Larghezza Lastra
																WorkPickPointOffset^[NPickPoint].Y;						// Valore di Offset Di Prelievo in Y
		3:	
			TFPalletizer_CalcolaCoordinataPrelievo_PickPoint := WorkPickPoint^[NPickPoint].Z +							// Quota Z, altezza della postazione
																WorkPickPointState^[NPickPoint].Element.ZDim +			// Metà Larghezza Lastra
																WorkPickPointOffset^[NPickPoint].Z;						// Valore di Offset Di Prelievo in Y
		4:	
			TFPalletizer_CalcolaCoordinataPrelievo_PickPoint := WorkPickPoint^[NPickPoint].J +							// Quota Y centro Rulliera	
																WorkPickPointOffset^[NPickPoint].J;						// Valore di Offset Di Prelievo in Y	
	END_CASE
ELSE
	CASE Ncase OF
		1:
			//TFPalletizer_CalcolaCoordinataPrelievo_PickPoint := WorkPickPoint^[NPickPoint].X +							// Quota X centro Rulliera	
			//													//WorkPickPointState^[NPickPoint].XPosBandella +	// Quota Relativa della posizione della bandella
			//													//(WorkPickPointState^[NPickPoint].Element.XDim/2) +		// Metà Lunghezza Lastra
			//													WorkPickPointOffset^[NPickPoint].X;						// Valore di Offset Di Prelievo in X	
		
			CASE TIPOLOGIA_RULLIERA_PRELIEVO OF
					
				RULLIERA_LONGITUDINALE:
										TFPalletizer_CalcolaCoordinataPrelievo_PickPoint := WorkPickPoint^[NPickPoint].X -							// Quota X centro Rulliera	
																//WorkPickPointState^[NPickPoint].XPosBandella +	// Quota Relativa della posizione della bandella
																//(WorkPickPointState^[NPickPoint].Element.XDim/2) +		// Metà Lunghezza Lastra
																MAX(Dimensioni_Pinza.Lunghezza/2,WorkPickPointState^[NPickPoint].Element.XDim/2) +
																WorkPickPointOffset^[NPickPoint].X;						// Valore di Offset Di Prelievo in X	
		
					
				RULLIERA_TRASVERSALE:
										TFPalletizer_CalcolaCoordinataPrelievo_PickPoint := WorkPickPoint^[NPickPoint].X +							// Quota X centro Rulliera	
																//WorkPickPointState^[NPickPoint].XPosBandella +	// Quota Relativa della posizione della bandella
																//(WorkPickPointState^[NPickPoint].Element.XDim/2) +		// Metà Lunghezza Lastra
																WorkPickPointOffset^[NPickPoint].X;						// Valore di Offset Di Prelievo in X	
									
			END_CASE
													
		2:	
			//TFPalletizer_CalcolaCoordinataPrelievo_PickPoint := WorkPickPoint^[NPickPoint].Y -							// Quota Y centro Rulliera	
			//												//	WorkPickPointState^[NPickPoint].YPosBandella +	// Quota Relativa della posizione della bandella
			//													(WorkPickPointState^[NPickPoint].Element.YDim/2) +		// Metà Larghezza Lastra
			//													WorkPickPointOffset^[NPickPoint].Y;						// Valore di Offset Di Prelievo in Y
	
			CASE TIPOLOGIA_RULLIERA_PRELIEVO OF
					
				RULLIERA_LONGITUDINALE:
										TFPalletizer_CalcolaCoordinataPrelievo_PickPoint := WorkPickPoint^[NPickPoint].Y +							// Quota Y centro Rulliera	
															//	WorkPickPointState^[NPickPoint].YPosBandella +	// Quota Relativa della posizione della bandella
															//	(WorkPickPointState^[NPickPoint].Element.YDim/2) +		// Metà Larghezza Lastra
																WorkPickPointOffset^[NPickPoint].Y;						// Valore di Offset Di Prelievo in Y
				RULLIERA_TRASVERSALE:
										TFPalletizer_CalcolaCoordinataPrelievo_PickPoint := WorkPickPoint^[NPickPoint].Y -							// Quota Y centro Rulliera	
															//	WorkPickPointState^[NPickPoint].YPosBandella +	// Quota Relativa della posizione della bandella
																(WorkPickPointState^[NPickPoint].Element.YDim/2) +		// Metà Larghezza Lastra
																WorkPickPointOffset^[NPickPoint].Y;						// Valore di Offset Di Prelievo in Y
				
			END_CASE


		3:	
			TFPalletizer_CalcolaCoordinataPrelievo_PickPoint := WorkPickPoint^[NPickPoint].Z +							// Quota Y centro Rulliera	
																WorkPickPointState^[NPickPoint].Element.ZDim +			// Metà Larghezza Lastra
																WorkPickPointOffset^[NPickPoint].Z;						// Valore di Offset Di Prelievo in Y
		4:	
			TFPalletizer_CalcolaCoordinataPrelievo_PickPoint := WorkPickPoint^[NPickPoint].J +							// Quota Y centro Rulliera	
																WorkPickPointOffset^[NPickPoint].J;						// Valore di Offset Di Prelievo in Y	
	END_CASE
END_IF

END_FUNCTION

// ---- POUs/TFPalletizerDataTF/Utility Varie/TFCalcoliIngombroPinza.TcPOU
(* Funzione che calcola l'ingombro della pinza nelle varie dimensioni a seconda del ciclo che la massima sta eseguendo *)
FUNCTION TFCalcoliIngombroPinza : BOOL
VAR_INPUT

	Mission : POINTER TO TFMachinePalletizer_Mission;
	WorkAreaManager : POINTER TO TFWorkAreaManager;
	WorkAreaState : POINTER TO ARRAY [1..MAXAREA] OF TFMachinePalletizer_WorkAreaState;

	AngoloRotazioneDestinazionePinza : LREAL; //Ango di rotazione del quale si vogliono calcolare le quote degli ingombri a destinazione  
	ModuleAX_J : POINTER TO TFModulePalletizer_AxJ_Lastre;//Modulo Asse rotazione
	
	IngombroX_Pos : POINTER TO LREAL;//Ingombro della pinza nella Metà POSITIVA della pinza lungo X
	IngombroY_Pos : POINTER TO LREAL;//Ingombro della pinza nella Metà POSITIVA della pinza lungo Y
	
	IngombroX_Neg : POINTER TO LREAL;//Ingombro della pinza nella Metà NEGATIVA della pinza lungo X
	IngombroY_Neg : POINTER TO LREAL;//Ingombro della pinza nella Metà NEGATIVA della pinza lungo Y
	
	IngombroY_Tot : POINTER TO LREAL;//Ingombro totale In direzione Y
	
	IngombroZ_Pos : POINTER TO LREAL;//Ingombro della pinza lungo Z Positivo (sopra al fulcro)
	IngombroZ_Neg : POINTER TO LREAL;//Ingombro della pinza lungo Z Negativo (sotto al fulcro)
	
	IngombroDestinazioneX_Pos : POINTER TO LREAL;//Ingombro della pinza nella Metà POSITIVA della pinza lungo X
	IngombroDestinazioneY_Pos : POINTER TO LREAL;//Ingombro della pinza nella Metà POSITIVA della pinza lungo Y
	
	IngombroDestinazioneX_Neg : POINTER TO LREAL;//Ingombro della pinza nella Metà NEGATIVA della pinza lungo X
	IngombroDestinazioneY_Neg : POINTER TO LREAL;//Ingombro della pinza nella Metà NEGATIVA della pinza lungo Y
	
	IngombroDestinazioneZ_Pos : POINTER TO LREAL;//Ingombro della pinza lungo Z Positivo (sopra al fulcro)
	IngombroDestinazioneZ_Neg : POINTER TO LREAL;//Ingombro della pinza lungo Z Negativo (sotto al fulcro)
	
	IngombroMaxX_Pos : POINTER TO LREAL;//Ingombro MASSIMO della pinza nella Metà POSITIVA della pinza lungo X
	IngombroMaxY_Pos : POINTER TO LREAL;//Ingombro MASSIMO della pinza nella Metà POSITIVA della pinza lungo Y
	
	IngombroMaxX_Neg : POINTER TO LREAL;//Ingombro MASSIMO della pinza nella Metà NEGATIVA della pinza lungo X
	IngombroMaxY_Neg : POINTER TO LREAL;//Ingombro MASSIMO della pinza nella Metà NEGATIVA della pinza lungo Y
	
	IngombroMaxZ_Pos : POINTER TO LREAL;//Ingombro MASSIMO della pinza lungo Z Positivo (sopra al fulcro)
	IngombroMaxZ_Neg : POINTER TO LREAL;//Ingombro MASSIMO della pinza lungo Z Negativo (sotto al fulcro)

	IngombroY_Pos_0 	: POINTER TO LREAL;//Ingombro della pinza nella Metà POSITIVA della pinza lungo Y nella posizione 0°
	IngombroY_Neg_180 	: POINTER TO LREAL;//Ingombro della pinza nella Metà NEGATIVA della pinza lungo Y nella posizione 180°
	IngombroY_Neg_0 	: POINTER TO LREAL;//Ingombro della pinza nella Metà POSITIVA della pinza lungo Y nella posizione 0°
	IngombroY_Pos_180 	: POINTER TO LREAL;//Ingombro della pinza nella Metà NEGATIVA della pinza lungo Y nella posizione 180°
	
	ScostamentoVerticalePuntoCentrale : POINTER TO LREAL; //Valore che rappresenta quanto il punto centrale si è spostato rispetto allo zero orizzontale (lungo Z crescente)
END_VAR

VAR
	LunghezzaMAX 	: LREAL;//LunghezzaMAX Totale pinza
	LarghezzaMAX 	: LREAL;//Larghezza Totale pinza
	SpessoreMAX  	: LREAL;//Spessore Totale pinza	
	DimTraveVerticale : LREAL; //Dimensione Trave/Ingombro Centrale
	
END_VAR

(* Calcolo delle dimensioni della pinza in base al tipo di ciclo in corso *)

CASE WorkAreaManager^.State OF
	WAMANAGER_NOP,
	
	WAMANAGER_CICLO_RIPOSO_INIT:
		SpessoreMAX 	:= Dimensioni_Pinza.Spessore;
		LunghezzaMAX 	:= Dimensioni_Pinza.Lunghezza;
		LarghezzaMAX    := Dimensioni_Pinza.Larghezza;
		
	WAMANAGER_CICLO_RIPOSO_RUN:
		
		SpessoreMAX 	:= Dimensioni_Pinza.Spessore;
		LunghezzaMAX 	:= Dimensioni_Pinza.Lunghezza;
		LarghezzaMAX    := Dimensioni_Pinza.Larghezza;
															
	WAMANAGER_CICLO_PRELIEVO_FALDA_RUN:
	
		SpessoreMAX 	:= Dimensioni_Pinza.Spessore;
		LunghezzaMAX 	:= Dimensioni_Pinza.Lunghezza;
		LarghezzaMAX    := Dimensioni_Pinza.Larghezza;

	WAMANAGER_CICLO_DEPOSITO_FALDA_RUN:
		
		SpessoreMAX 	:= Dimensioni_Pinza.Spessore;
		LunghezzaMAX 	:= MAX(Dimensioni_Pinza.Lunghezza,Mission^.XDim);
		LarghezzaMAX    := MAX(Dimensioni_Pinza.Larghezza,Mission^.YDim);

	WAMANAGER_CICLO_LASTRA_WA_INIT:
		SpessoreMAX 	:= Dimensioni_Pinza.Spessore;
		LunghezzaMAX 	:= MAX(Dimensioni_Pinza.Lunghezza,Mission^.XDim);
		LarghezzaMAX    := MAX(Dimensioni_Pinza.Larghezza,Mission^.YDim);
										
	WAMANAGER_CICLO_PRELIEVO_LASTRA_WA_RUN:
		SpessoreMAX 	:= Dimensioni_Pinza.Spessore;
		LunghezzaMAX 	:= Dimensioni_Pinza.Lunghezza;
		LarghezzaMAX    := Dimensioni_Pinza.Larghezza;
					
	WAMANAGER_CICLO_DEPOSITO_LASTRA_SU_PAREGGIATORE_RUN:
		SpessoreMAX 	:= Dimensioni_Pinza.Spessore;
		LunghezzaMAX 	:= MAX(Dimensioni_Pinza.Lunghezza,Mission^.XDim);
		LarghezzaMAX    := MAX(Dimensioni_Pinza.Larghezza,Mission^.YDim);
					
	WAMANAGER_CICLO_PRELIEVO_LASTRA_DA_PAREGGIATORE_RUN:
	
		SpessoreMAX 	:= Dimensioni_Pinza.Spessore;
		LunghezzaMAX 	:= Dimensioni_Pinza.Lunghezza;
		LarghezzaMAX    := Dimensioni_Pinza.Larghezza;
								
	WAMANAGER_CICLO_DEPOSITO_LASTRA_WA_RUN:
	
		SpessoreMAX 	:= Dimensioni_Pinza.Spessore;
		LunghezzaMAX 	:= MAX(Dimensioni_Pinza.Lunghezza,Mission^.XDim);
		LarghezzaMAX    := MAX(Dimensioni_Pinza.Larghezza,Mission^.YDim);

	WAMANAGER_CICLO_LASTRA_PP_INIT:
		SpessoreMAX 	:= Dimensioni_Pinza.Spessore;
		LunghezzaMAX 	:= Dimensioni_Pinza.Lunghezza;
		LarghezzaMAX    := Dimensioni_Pinza.Larghezza;
						
	WAMANAGER_CICLO_PRELIEVO_LASTRA_PP_RUN:
	
		SpessoreMAX 	:= Dimensioni_Pinza.Spessore;
		LunghezzaMAX 	:= Dimensioni_Pinza.Lunghezza;
		LarghezzaMAX    := Dimensioni_Pinza.Larghezza;
						
	WAMANAGER_CICLO_DEPOSITO_LASTRA_PP_RUN:
	
		SpessoreMAX 	:= Dimensioni_Pinza.Spessore;
		LunghezzaMAX 	:= MAX(Dimensioni_Pinza.Lunghezza,Mission^.XDim);
		LarghezzaMAX    := MAX(Dimensioni_Pinza.Larghezza,Mission^.YDim);

	(* Ciclo lastra per depalettizzare da postazioni senza formature, con autoapprndimenti*)
	WAMANAGER_CICLO_PRELIEVO_LASTRA_DEPAL_RUN :
	
		SpessoreMAX 	:= Dimensioni_Pinza.Spessore;
		LunghezzaMAX 	:= Dimensioni_Pinza.Lunghezza;
		LarghezzaMAX    := Dimensioni_Pinza.Larghezza;
																				
	(* Ciclo lastra deposito su rulliera *)
	WAMANAGER_CICLO_DEPOSITO_LASTRA_DEPAL_RUN :
	
		SpessoreMAX 	:= Dimensioni_Pinza.Spessore;
		LunghezzaMAX 	:= MAX(Dimensioni_Pinza.Lunghezza,Mission^.XDim);
		LarghezzaMAX    := MAX(Dimensioni_Pinza.Larghezza,Mission^.YDim);
													
	(* Ciclo deposito FALDA su magazzino dedicato *)
	WAMANAGER_CICLO_DEPOSITO_FALDA_DEPAL_RUN :
	
		SpessoreMAX 	:= Dimensioni_Pinza.Spessore;
		LunghezzaMAX 	:= MAX(Dimensioni_Pinza.Lunghezza,Mission^.XDim);
		LarghezzaMAX    := MAX(Dimensioni_Pinza.Larghezza,Mission^.YDim);
ELSE
		SpessoreMAX 	:= Dimensioni_Pinza.Spessore;
		LunghezzaMAX 	:= MAX(Dimensioni_Pinza.Lunghezza,Mission^.XDim);
		LarghezzaMAX    := MAX(Dimensioni_Pinza.Larghezza,Mission^.YDim);				
END_CASE

DimTraveVerticale := Dimensioni_Pinza.DimTraveVerticale;

(* Calcolo gli ingombri in base al'angolo di rotazione della pinza *)
IngombroX_Pos^ 	:=  LunghezzaMAX/2;
IngombroX_Neg^ 	:=  LunghezzaMAX/2;

IngombroY_Neg^ 	:= MAX((LarghezzaMAX/2 * COS(deg_to_rad(-90+ModuleAX_J^.Ax^.AxRef^.NcToPlc.ActPos)) +
					SpessoreMAX * SIN(deg_to_rad(-90+ModuleAX_J^.Ax^.AxRef^.NcToPlc.ActPos))),DimTraveVerticale/2);
					
IngombroY_Pos^ 	:= ABS(MIN((-LarghezzaMAX/2 * COS(deg_to_rad(-90+ModuleAX_J^.Ax^.AxRef^.NcToPlc.ActPos)) +
					SpessoreMAX * SIN(deg_to_rad(-90+ModuleAX_J^.Ax^.AxRef^.NcToPlc.ActPos))),DimTraveVerticale/2));	

(* In base a come la pinza è ruotata inverto il positivo con il negativo in modo da avere sempre i valori corretti *)
IF AngoloRotazioneDestinazionePinza < 90 THEN	                         
	IngombroZ_Pos^	:= ABS(((LarghezzaMAX/2) * SIN(deg_to_rad(-90+ModuleAX_J^.Ax^.AxRef^.NcToPlc.ActPos)))+
									(SpessoreMAX * COS(deg_to_rad(-90+ModuleAX_J^.Ax^.AxRef^.NcToPlc.ActPos)))-SpessoreMAX);

	IngombroZ_Neg^	:= ABS((-(LarghezzaMAX/2) * SIN(deg_to_rad(-90+ModuleAX_J^.Ax^.AxRef^.NcToPlc.ActPos))) +
									(SpessoreMAX * COS(deg_to_rad(-90+ModuleAX_J^.Ax^.AxRef^.NcToPlc.ActPos)))-SpessoreMAX);

ELSIF  AngoloRotazioneDestinazionePinza > 90 THEN					
	IngombroZ_Pos^	:= ABS((-(LarghezzaMAX/2) * SIN(deg_to_rad(-90+ModuleAX_J^.Ax^.AxRef^.NcToPlc.ActPos))) +
									(SpessoreMAX * COS(deg_to_rad(-90+ModuleAX_J^.Ax^.AxRef^.NcToPlc.ActPos)))-SpessoreMAX);	
	(*IngombroZ_Neg^	:= ABS(((LarghezzaMAX/2) * SIN(deg_to_rad(-90+ModuleAX_J^.Ax^.AxRef^.NcToPlc.ActPos)))+
								(SpessoreMAX * COS(deg_to_rad(-90+ModuleAX_J^.Ax^.AxRef^.NcToPlc.ActPos)))-SpessoreMAX); *)
	IngombroZ_Neg^	:= ABS((-(LarghezzaMAX/2) * SIN(deg_to_rad(-90+ModuleAX_J^.Ax^.AxRef^.NcToPlc.ActPos)))+
								(SpessoreMAX * COS(deg_to_rad(-90+ModuleAX_J^.Ax^.AxRef^.NcToPlc.ActPos)))-SpessoreMAX);
ELSE
	IngombroZ_Pos^	:= ABS(((LarghezzaMAX/2) * SIN(deg_to_rad(-90+ModuleAX_J^.Ax^.AxRef^.NcToPlc.ActPos)))+
									(SpessoreMAX * COS(deg_to_rad(-90+ModuleAX_J^.Ax^.AxRef^.NcToPlc.ActPos)))-SpessoreMAX);

	IngombroZ_Neg^	:= ABS((-(LarghezzaMAX/2) * SIN(deg_to_rad(-90+ModuleAX_J^.Ax^.AxRef^.NcToPlc.ActPos))) +
									(SpessoreMAX * COS(deg_to_rad(-90+ModuleAX_J^.Ax^.AxRef^.NcToPlc.ActPos)))-SpessoreMAX);
END_IF
IngombroY_Tot := IngombroY_Pos + IngombroY_Neg;//Ingombro TOTALE in direzione Y


(* Calcolo gli ingombri in base al'angolo di rotazione FINALE *)
IngombroDestinazioneX_Pos^ 	:=  LunghezzaMAX/2;
IngombroDestinazioneX_Neg^ 	:=  LunghezzaMAX/2;

IngombroDestinazioneY_Neg^ 	:= MAX((LarghezzaMAX/2 * COS(deg_to_rad(-90+AngoloRotazioneDestinazionePinza)) +
									SpessoreMAX * SIN(deg_to_rad(-90+AngoloRotazioneDestinazionePinza))),DimTraveVerticale/2);
					
IngombroDestinazioneY_Pos^ 	:= ABS(MIN((-LarghezzaMAX/2 * COS(deg_to_rad(-90+AngoloRotazioneDestinazionePinza)) +
									SpessoreMAX * SIN(deg_to_rad(-90+AngoloRotazioneDestinazionePinza))),DimTraveVerticale/2));
	
(* In base a come la pinza è ruotata inverto il positivo con il negativo in modo da avere sempre i valori corretti *)
IF AngoloRotazioneDestinazionePinza < 90 THEN	                         
	IngombroDestinazioneZ_Pos^	:= ABS(((LarghezzaMAX/2) * SIN(deg_to_rad(-90+AngoloRotazioneDestinazionePinza)))+
									(SpessoreMAX * COS(deg_to_rad(-90+AngoloRotazioneDestinazionePinza)))-SpessoreMAX);

	IngombroDestinazioneZ_Neg^	:= ABS((-(LarghezzaMAX/2) * SIN(deg_to_rad(-90+AngoloRotazioneDestinazionePinza))) +
									(SpessoreMAX * COS(deg_to_rad(-90+AngoloRotazioneDestinazionePinza)))-SpessoreMAX);

ELSIF  AngoloRotazioneDestinazionePinza > 90.9 THEN		
	//AlPosDestinoBandelCavaleta := Mission^.YDim / 2 + WorkAreaState^[Mission^.PPlace].Supporto.ZDim + WorkAreaState^[Mission^.PPick].Supporto.HMAX;			
	IngombroDestinazioneZ_Pos^	:= ABS((-(LarghezzaMAX/2) * SIN(deg_to_rad(-90+AngoloRotazioneDestinazionePinza))) +
									(SpessoreMAX * COS(deg_to_rad(-90+AngoloRotazioneDestinazionePinza)))-SpessoreMAX);	
	IngombroDestinazioneZ_Neg^	:= ABS(((LarghezzaMAX/2) * SIN(deg_to_rad(-90+AngoloRotazioneDestinazionePinza)))+
								(SpessoreMAX * COS(deg_to_rad(-90+AngoloRotazioneDestinazionePinza)))-SpessoreMAX) ;
	
	
ELSE
	IngombroDestinazioneZ_Pos^	:= ABS(((LarghezzaMAX/2) * SIN(deg_to_rad(-90+AngoloRotazioneDestinazionePinza)))+
									(SpessoreMAX * COS(deg_to_rad(-90+AngoloRotazioneDestinazionePinza)))-SpessoreMAX);

	IngombroDestinazioneZ_Neg^	:= ABS((-(LarghezzaMAX/2) * SIN(deg_to_rad(-90+AngoloRotazioneDestinazionePinza))) +
									(SpessoreMAX * COS(deg_to_rad(-90+AngoloRotazioneDestinazionePinza)))-SpessoreMAX);
END_IF

(* Calcolo degli ingombri massimi nelle varie dimensioni *)
IngombroMaxX_Pos^ := MAX(IngombroX_Pos^,IngombroDestinazioneX_Pos^);//Ingombro MASSIMO della pinza nella Metà POSITIVA della pinza lungo X
IngombroMaxY_Pos^ := MAX(IngombroY_Pos^,IngombroDestinazioneY_Pos^);//Ingombro MASSIMO della pinza nella Metà POSITIVA della pinza lungo Y

IngombroMaxX_Neg^ := MAX(IngombroX_Neg^,IngombroDestinazioneX_Neg^);//Ingombro MASSIMO della pinza nella Metà NEGATIVA della pinza lungo X
IngombroMaxY_Neg^ := MAX(IngombroY_Neg^,IngombroDestinazioneY_Neg^);//Ingombro MASSIMO della pinza nella Metà NEGATIVA della pinza lungo Y

IngombroMaxZ_Pos^ := MAX(IngombroZ_Pos^,IngombroDestinazioneZ_Pos^);//Ingombro MASSIMO della pinza lungo Z Positivo (sopra al fulcro)
IngombroMaxZ_Neg^ := MAX(IngombroZ_Neg^,IngombroDestinazioneZ_Neg^);//Ingombro MASSIMO della pinza lungo Z Negativo (sotto al fulcro)

//IngombroMaxZ_Pos^ := MIN( MAX(IngombroZ_Pos^,IngombroDestinazioneZ_Pos^),(LarghezzaMAX/2)+ SpessoreMAX);//Ingombro MASSIMO della pinza lungo Z Positivo (sopra al fulcro)
//IngombroMaxZ_Neg^ := MIN( MAX(IngombroZ_Neg^,IngombroDestinazioneZ_Neg^),(LarghezzaMAX/2)+ SpessoreMAX);//Ingombro MASSIMO della pinza lungo Z Negativo (sotto al fulcro)




/////////////////////////////

IngombroY_Pos_0^ := ABS(MIN(SpessoreMAX * SIN(deg_to_rad(-90)),DimTraveVerticale/2));
IngombroY_Neg_180^ := ABS(MAX(SpessoreMAX * SIN(deg_to_rad(-90+180)),DimTraveVerticale/2));

IngombroY_Neg_0^ := ABS(MAX(SpessoreMAX * SIN(deg_to_rad(-90)),DimTraveVerticale/2));
IngombroY_Pos_180^ := ABS(MIN(SpessoreMAX * SIN(deg_to_rad(-90+180)),DimTraveVerticale/2));
								
ScostamentoVerticalePuntoCentrale^ := ABS(SpessoreMAX * COS(deg_to_rad(-90+AngoloRotazioneDestinazionePinza))-SpessoreMAX);
																
TFCalcoliIngombroPinza := TRUE;

END_FUNCTION

// ---- Data types/AlbertoPruevas/Funciones/FunLadoTrabajoCaballete.TcPOU
FUNCTION FunLadoTrabajoCaballete : Uint
VAR_INPUT
	Piezas_LadoA 			: UINT ;
	Piezas_Ladob			: UINT ;
	Recoger					: BOOL;
	Dejar					: BOOL ;
	GestionLadoTrabajo		: INT ;
	//Tiporecogida			: UINT;
	GestionDescargaCaballete			: POINTER TO Es_LadosCaballete ;
END_VAR
VAR
	DifPiezas 				: UINT;
	Piezas_ladoAdif			: UINT;
	Piezas_ladoBdif			: UINT;
END_VAR

IF  Dejar AND GestionLadoTrabajo = 0 THEN 
  
	IF Piezas_LadoA = 0 AND Piezas_Ladob =0 THEN 
		FunLadoTrabajoCaballete := 0 ;
	
	ELSIF Piezas_LadoA <> Piezas_Ladob THEN 
		DifPiezas := ABS (Piezas_LadoA - Piezas_Ladob) ;
			IF DifPiezas > 1 AND Piezas_LadoA > Piezas_Ladob THEN 
				FunLadoTrabajoCaballete := 180 ;
			ELSIF DifPiezas > 1 AND Piezas_Ladob > Piezas_LadoA	THEN
				FunLadoTrabajoCaballete := 0 ;
			END_IF
	END_IF
		
	IF DifPiezas = 1   THEN
			IF  Piezas_Ladob < Piezas_LadoA THEN 
				FunLadoTrabajoCaballete := 180 ;
			ELSIF Piezas_LadoA < Piezas_LadoB THEN 
				FunLadoTrabajoCaballete := 0 ;
			END_IF
	END_IF
END_IF

IF  Recoger AND GestionLadoTrabajo = 0  THEN 
	IF Piezas_LadoA <> Piezas_Ladob AND GestionDescargaCaballete^.Lado_trabajo = E_Ul_RecogidaCaballete.Primera_Pieza  THEN 
		GestionDescargaCaballete^.TipoRecogida := 1 ;
		IF Piezas_LadoA > Piezas_Ladob THEN 
			IF Piezas_Ladob > 0 THEN
				GestionDescargaCaballete^.Dif_PiezasLados := Piezas_LadoA - Piezas_Ladob;
			ELSE 
				GestionDescargaCaballete^.Dif_PiezasLados := 0 ;	
			END_IF
			GestionDescargaCaballete^.Lado_trabajo := E_Ul_RecogidaCaballete.LadoAMayor ;
		ELSIF Piezas_Ladob > Piezas_LadoA THEN 
			IF Piezas_LadoA > 0 THEN 
				GestionDescargaCaballete^.Dif_PiezasLados := Piezas_Ladob - Piezas_LadoA;
			ELSE
				GestionDescargaCaballete^.Dif_PiezasLados := 0 ;	
			END_IF 
			GestionDescargaCaballete^.Lado_trabajo := E_Ul_RecogidaCaballete.LadoBMayor ;	
		END_IF
	ELSIF Piezas_LadoA = Piezas_Ladob AND GestionDescargaCaballete^.Lado_trabajo = E_Ul_RecogidaCaballete.Primera_Pieza THEN 
		GestionDescargaCaballete^.TipoRecogida := 0 ;
		GestionDescargaCaballete^.Dif_PiezasLados := 0;
	END_IF 	

	IF GestionDescargaCaballete^.TipoRecogida = 1  THEN
		IF GestionDescargaCaballete^.Lado_trabajo = E_Ul_RecogidaCaballete.LadoAMayor THEN 
			Piezas_ladoAdif := Piezas_LadoA - GestionDescargaCaballete^.Dif_PiezasLados;
			Piezas_ladoBdif := Piezas_Ladob ;
		ELSIF GestionDescargaCaballete^.Lado_trabajo = E_Ul_RecogidaCaballete.LadoBMayor THEN
 			Piezas_ladoBdif := Piezas_Ladob  - GestionDescargaCaballete^.Dif_PiezasLados ;
			Piezas_ladoAdif := Piezas_LadoA ;	
		END_IF
	END_IF
	IF GestionDescargaCaballete^.TipoRecogida = 0 THEN
		Piezas_ladoAdif := Piezas_LadoA ;
		Piezas_ladoBdif := Piezas_Ladob ;
	END_IF
	
	


	IF GestionDescargaCaballete^.TipoRecogida >= 0 THEN 
			IF Piezas_ladoAdif = Piezas_ladoBdif AND  Piezas_ladoBdif > 0 AND Piezas_ladoAdif >0  THEN 
				FunLadoTrabajoCaballete := 180 ;
			ELSIF Piezas_ladoAdif <> Piezas_ladoBdif THEN 
				DifPiezas := ABS (Piezas_ladoAdif - Piezas_ladoBdif) ;
					IF DifPiezas > 1 AND Piezas_ladoAdif > Piezas_ladoBdif THEN 
						FunLadoTrabajoCaballete := 0 ;
					ELSIF DifPiezas > 1 AND Piezas_ladoBdif > Piezas_ladoAdif	THEN
						FunLadoTrabajoCaballete := 180 ;
					END_IF
			END_IF
			
			 
	
			IF DifPiezas = 1  THEN
					IF  Piezas_ladoBdif < Piezas_ladoAdif THEN 
						FunLadoTrabajoCaballete := 0 ;
					ELSIF Piezas_ladoAdif < Piezas_ladoBdif THEN 
						FunLadoTrabajoCaballete := 180 ;
					END_IF
			ELSIF	DifPiezas < 0  THEN	
				IF  Piezas_ladoAdif < 0 THEN 
						FunLadoTrabajoCaballete := 0 ;
					ELSIF Piezas_ladoBdif < 0 THEN 
						FunLadoTrabajoCaballete := 180 ;
					END_IF
					
			END_IF
	END_IF 
END_IF


IF GestionLadoTrabajo <> 0 THEN
	IF GestionLadoTrabajo = 1 THEN
		FunLadoTrabajoCaballete := 0 ;
	ELSIF GestionLadoTrabajo = 2 THEN 
		FunLadoTrabajoCaballete := 180 ;	
	END_IF
	


END_IF

END_FUNCTION

// ---- POUs/TFCicliDiLavoro/ProgrammiMovimento/TFProgramma_Ciclo_Riposo_Lastre.TcPOU
FUNCTION_BLOCK TFProgramma_Ciclo_Riposo_Lastre
VAR_INPUT
	X_Par : Ax_Program_Parameters; // Parametri degli assi
	Y_Par : Ax_Program_Parameters; // Parametri degli assi
	Z_Par : Ax_Program_Parameters; // Parametri degli assi
	//K_Par : Ax_Program_Parameters; // Parametri degli assi
	J_Par : Ax_Program_Parameters; // Parametri degli assi
	
	(*X*)
	Quota_Riposo_X 	: LREAL;
	Quota_Fuori_Ingombro_X : LREAL;
	(*Y*)
	Quota_Riposo_Y	: LREAL;
	Quota_Fuori_Ingombro_Y : LREAL;
	(*Z*)
	Quota_Riposo_Z	: LREAL;
	Quota_Fuori_Ingombro_Z : LREAL;

	(*J*)
	Quota_Riposo_J	: LREAL;
	Quota_Fuori_Ingombro_J : LREAL;
END_VAR
VAR_OUTPUT
	Inizializzato : BOOL;
END_VAR
VAR
	;
END_VAR

(* CICLO DI RIPOSO *)
Inizializzato := FALSE;
(*************************************************************************************************************************************)
(******************************************************  ASSE X **********************************************************************)
(*************************************************************************************************************************************)
(* Programma 0 Asse X : Traslazione a quota di riposo*)
Programma_X[0].ID 					:= 0;
Programma_X[0].Quota_Destinazione	:= Quota_Riposo_X;
Programma_X[0].Velocita				:= X_Par.Vel_Vuoto;
Programma_X[0].Accelerazione		:= X_Par.Acc_Vuoto;
Programma_X[0].Decelerazione		:= X_Par.Dec_Vuoto;
Programma_X[0].Jerk					:= X_Par.Jerk_Vuoto;

(* Programma 6 Asse X : Traslazione a quota di FUORI INGOMBRO*)
Programma_X[6].ID 					:= 6;
Programma_X[6].Quota_Destinazione	:= Quota_Fuori_Ingombro_X;
Programma_X[6].Velocita				:= X_Par.Vel_Vuoto;
Programma_X[6].Accelerazione		:= X_Par.Acc_Vuoto;
Programma_X[6].Decelerazione		:= X_Par.Dec_Vuoto;
Programma_X[6].Jerk					:= X_Par.Jerk_Vuoto;

(*************************************************************************************************************************************)
(******************************************************  ASSE Y **********************************************************************)
(*************************************************************************************************************************************)
(* Programma 0 Asse Y : Traslazione a quota di riposo*)
Programma_Y[0].ID 					:= 0;
Programma_Y[0].Quota_Destinazione	:= Quota_Riposo_Y;
Programma_Y[0].Velocita				:= Y_Par.Vel_Vuoto;
Programma_Y[0].Accelerazione		:= Y_Par.Acc_Vuoto;
Programma_Y[0].Decelerazione		:= Y_Par.Dec_Vuoto;
Programma_Y[0].Jerk					:= Y_Par.Jerk_Vuoto;

(* Programma 6 Asse Y : Traslazione a quota di FUORI INGOMBRO*)
Programma_Y[6].ID 					:= 6;
Programma_Y[6].Quota_Destinazione	:= Quota_Fuori_Ingombro_Y;
Programma_Y[6].Velocita				:= Y_Par.Vel_Vuoto;
Programma_Y[6].Accelerazione		:= Y_Par.Acc_Vuoto;
Programma_Y[6].Decelerazione		:= Y_Par.Dec_Vuoto;
Programma_Y[6].Jerk					:= Y_Par.Jerk_Vuoto;

(*************************************************************************************************************************************)
(******************************************************  ASSE Z **********************************************************************)
(*************************************************************************************************************************************)

(* Programma 0 Asse Z : Traslazione a quota di riposo*)
Programma_Z[0].ID 					:= 0;
Programma_Z[0].Quota_Destinazione	:= Quota_Riposo_Z;
Programma_Z[0].Velocita				:= Z_Par.Vel_Vuoto;
Programma_Z[0].Accelerazione		:= Z_Par.Acc_Vuoto;
Programma_Z[0].Decelerazione		:= Z_Par.Dec_Vuoto;
Programma_Z[0].Jerk					:= Z_Par.Jerk_Vuoto;
Programma_Z[0].DisabilitaTasteggio	:= TRUE;

(* Programma 6 Asse Z : Traslazione a quota di FUORI INGOMBRO*)
Programma_Z[6].ID 					:= 6;
Programma_Z[6].Quota_Destinazione	:= Quota_Fuori_Ingombro_Z;
Programma_Z[6].Velocita				:= Z_Par.Vel_Vuoto;
Programma_Z[6].Accelerazione		:= Z_Par.Acc_Vuoto;
Programma_Z[6].Decelerazione		:= Z_Par.Dec_Vuoto;
Programma_Z[6].Jerk					:= Z_Par.Jerk_Vuoto;
Programma_Z[6].DisabilitaTasteggio	:= TRUE;

(*
(*************************************************************************************************************************************)
(******************************************************  ASSE K **********************************************************************)
(*************************************************************************************************************************************)

(* Programma 0 Asse K : Traslazione a quota di ripos *)
Programma_K[0].ID 					:= 0;
Programma_K[0].Quota_Destinazione	:= Quota_Riposo_K;
Programma_K[0].Velocita				:= K_Par.Vel_Vuoto;
Programma_K[0].Accelerazione		:= K_Par.Acc_Vuoto;
Programma_K[0].Decelerazione		:= K_Par.Dec_Vuoto;
Programma_K[0].Jerk					:= K_Par.Jerk_Vuoto;
Programma_K[0].Torque				:= 100;
Programma_K[0].ControlloCoppiaAbilitato := FALSE;
Programma_K[0].Controllo_Tastatori	:= TRUE;
*)
(*************************************************************************************************************************************)
(******************************************************  ASSE J **********************************************************************)
(*************************************************************************************************************************************)

(* Programma 0 Asse J : Traslazione a quota di riposo *)
Programma_J[0].ID 					:= 0;
Programma_J[0].Quota_Destinazione	:= Quota_Riposo_J;
Programma_J[0].Velocita				:= J_Par.Vel_Vuoto;
Programma_J[0].Accelerazione		:= J_Par.Acc_Vuoto;
Programma_J[0].Decelerazione		:= J_Par.Dec_Vuoto;
Programma_J[0].Jerk					:= J_Par.Jerk_Vuoto;

(* Programma 6 Asse Z : Traslazione a quota di FUORI INGOMBRO*)
Programma_J[6].ID 					:= 6;
Programma_J[6].Quota_Destinazione	:= Quota_Fuori_Ingombro_J;
Programma_J[6].Velocita				:= J_Par.Vel_Vuoto;
Programma_J[6].Accelerazione		:= J_Par.Acc_Vuoto;
Programma_J[6].Decelerazione		:= J_Par.Dec_Vuoto;
Programma_J[6].Jerk					:= J_Par.Jerk_Vuoto;
Programma_J[6].DisabilitaTasteggio	:= TRUE;

(* Programma 6 Asse J : Traslazione a quota di FUORI INGOMBRO*)
Programma_J[J_PosFuoriIngombro].ID 					:= TO_UINT(J_PosFuoriIngombro);
Programma_J[J_PosFuoriIngombro].Quota_Destinazione	:= Quota_Fuori_Ingombro_J;
Programma_J[J_PosFuoriIngombro].Velocita			:= J_Par.Vel_Vuoto;
Programma_J[J_PosFuoriIngombro].Accelerazione		:= J_Par.Acc_Vuoto;
Programma_J[J_PosFuoriIngombro].Decelerazione		:= J_Par.Dec_Vuoto;
Programma_J[J_PosFuoriIngombro].Jerk				:= J_Par.Jerk_Vuoto;
Programma_J[J_PosFuoriIngombro].DisabilitaTasteggio	:= TRUE;

Inizializzato := TRUE;

END_FUNCTION_BLOCK

// ---- POUs/TFCicliDiLavoro/ProgrammiMovimento/TFProgramma_Ciclo_Falda_Lastre.TcPOU
FUNCTION_BLOCK TFProgramma_Ciclo_Falda_Lastre
VAR_INPUT
	X_Par : Ax_Program_Parameters; // Parametri degli assi
	Y_Par : Ax_Program_Parameters; // Parametri degli assi
	Z_Par : Ax_Program_Parameters; // Parametri degli assi
	//K_Par : Ax_Program_Parameters; // Parametri degli assi
	J_Par : Ax_Program_Parameters; // Parametri degli assi
	
